// TwinCAT 3 PLC project TE1108
// ProgramVersion: 3.1.4026.22
// libraries:
//   Tc2_EtherCAT, * (Beckhoff Automation GmbH)
//   Tc2_IoFunctions, * (Beckhoff Automation GmbH)
//   Tc2_Standard, * (Beckhoff Automation GmbH)
//   Tc2_System, * (Beckhoff Automation GmbH)
//   Tc2_Utilities, * (Beckhoff Automation GmbH)
//   Tc3_Module, * (Beckhoff Automation GmbH)
// project tree:
//   DUTs/COMPONENTS/GENERIC/ ST_GeneralStationCMD.TcDUT (not stored), ST_StationStatus.TcDUT (not stored)
//   DUTs/COMPONENTS/HEIGHT TEST/ ST_HeightTest.TcDUT (not stored), ST_HeightTest_CMD.TcDUT (not stored), ST_ProbesSettings.TcDUT, E_HeightTest_State.TcDUT (not stored), ST_HeightTest_CycleData.TcDUT (not stored)
//   DUTs/COMPONENTS/LEAK TESTER/ ST_LeakTester.TcDUT (not stored), ST_LeakTester_CMD.TcDUT (not stored), E_LeakTester_State.TcDUT (not stored), ST_LeakTester_CycleData.TcDUT (not stored)
//   DUTs/COMPONENTS/MAIN CYLINDER/ ST_ProcessCylinder.TcDUT (not stored), E_ProcessCylinder_State.TcDUT (not stored), ST_ProcessCylinder_CMD.TcDUT (not stored)
//   DUTs/COMPONENTS/PROCESS DOOR/ E_ProcessDoor_State.TcDUT (not stored), ST_ProcessDoor.TcDUT (not stored), ST_ProcessDoor_CMD.TcDUT (not stored)
//   DUTs/COMPONENTS/SLIDE NEST/ E_SlideNest_State.TcDUT (not stored), ST_SlideNest.TcDUT (not stored), ST_SlideNest_CMD.TcDUT (not stored)
//   DUTs/HMI/ ST_Animations.TcDUT (not stored), ST_StatisticsHMI.TcDUT (not stored), ST_StatusBanner.TcDUT (not stored), ST_Timers.TcDUT (not stored)
//   DUTs/IO/CARDS/ ST_EL1918_C.TcDUT (not stored), ST_EL3058.TcDUT (not stored), ST_EL1918_A.TcDUT (not stored), ST_EL1918_B.TcDUT (not stored), ST_EL2904.TcDUT (not stored), ST_EL6910.TcDUT (not stored), ST_EL6633.TcDUT (not stored), ST_EL9410.TcDUT (not stored), ST_K1100.TcDUT (not stored), ST_EL6070.TcDUT (not stored), ST_Terminal_Info.TcDUT (not stored), ST_EL1809.TcDUT, ST_EL2809_A.TcDUT
//   DUTs/IO/LEAK_TESTERS/ ST_General_LeakTester_I_O.TcDUT (not stored), st_i28General_I_O.TcDUT (not stored), st_i28LasResult.TcDUT (not stored), st_i28LiveMeasurement.TcDUT (not stored)
//   DUTs/IO/PROBES/ ST_ProbesSet.TcDUT (not stored), ST_Probes_I_O.TcDUT (not stored)
//   DUTs/MASTER/ E_MachineState.TcDUT (not stored), ST_ButtonsLamps.TcDUT (not stored), ST_MachineStatus.TcDUT (not stored), ST_MasterCTRL.TcDUT (not stored), ST_Puls.TcDUT (not stored)
//   DUTs/MASTER/log_CSV/ ST_TableCycleData.TcDUT (not stored), ST_UserLog.TcDUT (not stored), ST_CycleData.TcDUT (not stored)
//   DUTs/MASTER/PROCESS CYCLES/ E_General_ProcessCycle.TcDUT
//   DUTs/PDFMaker/ ST_EventsPDF.TcDUT (not stored), ST_EventsPdfConstants.TcDUT (not stored), ST_JavasCriptPDF.TcDUT (not stored), ST_PDFMaker.TcDUT (not stored)
//   DUTs/ ST_SafeOutputsReading.TcDUT (not stored), ST_TwinSAFE.TcDUT (not stored)
//   DUTs/USER_ALARMS_EVENTS/EVENTS/ ST_ActiveEvents.TcDUT (not stored), ST_EventsAssigment.TcDUT (not stored), ST_EventsAssigmentGeneral.TcDUT (not stored), ST_EventsHistory.TcDUT (not stored), ST_EVENT.TcDUT (not stored), ST_StationEvents.TcDUT (not stored)
//   DUTs/USER_ALARMS_EVENTS/ ST_UserLogHMI.TcDUT (not stored)
//   GVLs/ GVL_Constants.TcGVL (not stored), GVL_HMI.TcGVL, GVL_IO.TcGVL (not stored), GVL_Master.TcGVL, GVL_Persistent.TcGVL (not stored), GVL_Stations.TcGVL
//   / PlcTask.TcTTO (not stored)
//   POUs/A_MASTER/ A_1_PRG_Main_Master.TcPOU, A_2_PRG_MachineCtrl.TcPOU, A_3_PRG_FaultHandling.TcPOU
//   POUs/B_STATIONS/B_1_LEAK_TEST/ B_1_1_PRG_Master_Leak_Test.TcPOU
//   POUs/B_STATIONS/B_2_HEIGHT_TEST/ B_2_1_PRG_Master_Height_Test.TcPOU (not stored)
//   POUs/B_STATIONS/B_4_PROCESS_CYLINDER__SLIDE_DOOR_SLIDE_NEST/ B_4_1_PRG_Master_ProcessCylinder.TcPOU, B_4_2_PRG_Master_ProcessDoor.TcPOU, B_4_3_PRG_Master_SlideNest.TcPOU
//   POUs/C_HMI/ C_1_PRG_MainHMI.TcPOU
//   POUs/D_CSV/ D_1_PRG_CycleDataCSV.TcPOU (not stored)
//   POUs/ MAIN.TcPOU (not stored)
//   POUs/Utilities/ FB_EventsManager.TcPOU (not stored), FB_PDFMaker.TcPOU (not stored), FB_Scale.TcPOU (not stored), FB_UserLog.TcPOU (not stored), FB_Pulse.TcPOU (not stored), FB_TerminalInfo.TcPOU (not stored), FB_TimeControl.TcPOU (not stored), PRG_Puls.TcPOU (not stored)
// real-time tasks:
//   TASK PlcTask: cycle T#10ms, priority 20, ADS port 350
// I/O:
//   DEVICE Device1(EtherCAT), AmsNetId 192.168.7.156.4.1
//     Term 1 (EK1100) [EK1100 EtherCAT Coupler (2A E-Bus)]
//       Term 2 (EL6070-0033) [EL6070-0033 1Ch. Licence key terminal, individual licences]
//       Term 3 (EL6910) [EL6910, TwinSAFE PLC]
//       Term 4 (EL1918) [EL1918, 8Ch. Safety Input 24V, TwinSAFE]
//         modules: Module 1 (FSOE), Module 2 (FSLOGIC)
//       Term 5 (EL1918) [EL1918, 8Ch. Safety Input 24V, TwinSAFE]
//         modules: Module 1 (FSOE), Module 2 (FSLOGIC)
//       Term 6 (EL2904) [EL2904, 4 Ch. Safety Output 24V, 0.5A, TwinSAFE]
//         modules: Module 1 (FSOES), Module 2 (DO)
//       Term 7 (EL9410) [EL9410 E-Bus Power Supplier  (Diagnostics)]
//       Term 8 (EL1809) [EL1809 16Ch. Dig. Input 24V, 3ms]
//       Term 9 (EL2809) [EL2809 16Ch. Dig. Output 24V, 0.5A]
//       Term 10 (EL3058) [EL3058 8Ch. Ana. Input 4-20mA]
//       Term 11(EL1918) [EL1918, 8Ch. Safety Input 24V, TwinSAFE]
//         modules: Module 1 (FSOE), Module 2 (FSLOGIC)
//       Term 12 (EL6633) [EL6633 PROFINET IO Controller]
//       Term 13 (EL9011) [EL9011 End Terminal]
//     Box 21 (DL-EC1A) [DL-EC1A]
//   DEVICE Profinet1 (EL6633), AmsNetId 192.168.7.156.2.1
//     fpc1 [Cincinnati Test Systems 1-port Device 00210]
//       modules: Term 1 (DAP Module), Term 2 (PLC Input), Term 3 (PLC Output  )
//     fpc2 [Cincinnati Test Systems 1-port Device 00210]
//       modules: Term 4 (DAP Module), Term 5 (PLC Input), Term 6 (PLC Output  )
// variable links:
//   Device1(EtherCAT) <-> Device1(EtherCAT)/Term 1 (EK1100)/Term 11(EL1918)
//     Term 1 (EK1100)/Term 3 (EL6910)/ConnectionInputs/Message_38 TxPDO <-> Module 1 (FSOE)/FSoE Outputs/FSOE
//     Term 1 (EK1100)/Term 3 (EL6910)/ConnectionOutputs/Message_38 RxPDO <-> Module 1 (FSOE)/FSoE Inputs/FSOE
//   Device1(EtherCAT) <-> Device1(EtherCAT)/Term 1 (EK1100)/Term 4 (EL1918)
//     Term 1 (EK1100)/Term 3 (EL6910)/ConnectionInputs/Message_8 TxPDO <-> Module 1 (FSOE)/FSoE Outputs/FSOE
//     Term 1 (EK1100)/Term 3 (EL6910)/ConnectionOutputs/Message_8 RxPDO <-> Module 1 (FSOE)/FSoE Inputs/FSOE
//   Device1(EtherCAT) <-> Device1(EtherCAT)/Term 1 (EK1100)/Term 5 (EL1918)
//     Term 1 (EK1100)/Term 3 (EL6910)/ConnectionInputs/Message_9 TxPDO <-> Module 1 (FSOE)/FSoE Outputs/FSOE
//     Term 1 (EK1100)/Term 3 (EL6910)/ConnectionOutputs/Message_9 RxPDO <-> Module 1 (FSOE)/FSoE Inputs/FSOE
//   Device1(EtherCAT) <-> Device1(EtherCAT)/Term 1 (EK1100)/Term 6 (EL2904)
//     Term 1 (EK1100)/Term 3 (EL6910)/ConnectionInputs/Message_10 TxPDO <-> Module 1 (FSOES)/RxPDO/FSOE
//     Term 1 (EK1100)/Term 3 (EL6910)/ConnectionOutputs/Message_10 RxPDO <-> Module 1 (FSOES)/TxPDO/FSOE
//   TE1108/TE1108 Instance <-> Device1(EtherCAT)/Box 21 (DL-EC1A)
//     PlcTask Inputs/GVL_IO.Probes.bGeneralError <-> Status of System/Error Status
//     PlcTask Inputs/GVL_IO.Probes.stProbesSet[1].abProbeError[1] <-> ID01 Status/ID01 Error Status
//     PlcTask Inputs/GVL_IO.Probes.stProbesSet[1].abProbeError[2] <-> ID02 Status/ID02 Error Status
//     PlcTask Inputs/GVL_IO.Probes.stProbesSet[1].abProbeError[3] <-> ID03 Status/ID03 Error Status
//     PlcTask Inputs/GVL_IO.Probes.stProbesSet[1].abProbeError[4] <-> ID04 Status/ID04 Error Status
//     PlcTask Inputs/GVL_IO.Probes.stProbesSet[2].abProbeError[1] <-> ID05 Status/ID05 Error Status
//     PlcTask Inputs/GVL_IO.Probes.stProbesSet[2].abProbeError[2] <-> ID06 Status/ID06 Error Status
//     PlcTask Inputs/GVL_IO.Probes.stProbesSet[2].abProbeError[3] <-> ID07 Status/ID07 Error Status
//     PlcTask Inputs/GVL_IO.Probes.stProbesSet[2].abProbeError[4] <-> ID08 Status/ID08 Error Status
//     PlcTask Inputs/GVL_IO.Probes.stProbesSet[1].anRawMeasurement[1] <-> ID01 Current Value/ID01 Current Value (P.V.)
//     PlcTask Inputs/GVL_IO.Probes.stProbesSet[1].anRawMeasurement[2] <-> ID02 Current Value/ID02 Current Value (P.V.)
//     PlcTask Inputs/GVL_IO.Probes.stProbesSet[1].anRawMeasurement[3] <-> ID03 Current Value/ID03 Current Value (P.V.)
//     PlcTask Inputs/GVL_IO.Probes.stProbesSet[1].anRawMeasurement[4] <-> ID04 Current Value/ID04 Current Value (P.V.)
//     PlcTask Inputs/GVL_IO.Probes.stProbesSet[2].anRawMeasurement[1] <-> ID05 Current Value/ID05 Current Value (P.V.)
//     PlcTask Inputs/GVL_IO.Probes.stProbesSet[2].anRawMeasurement[2] <-> ID06 Current Value/ID06 Current Value (P.V.)
//     PlcTask Inputs/GVL_IO.Probes.stProbesSet[2].anRawMeasurement[3] <-> ID07 Current Value/ID07 Current Value (P.V.)
//     PlcTask Inputs/GVL_IO.Probes.stProbesSet[2].anRawMeasurement[4] <-> ID08 Current Value/ID08 Current Value (P.V.)
//     PlcTask Inputs/GVL_IO.Probes.stTerminalInfo.nTerminal_State <-> InfoData/State
//     PlcTask Outputs/GVL_IO.Probes.abPresetProbe <-> Input Request 1/Request 1
//   TE1108/TE1108 Instance <-> Device1(EtherCAT)/Term 1 (EK1100)
//     PlcTask Inputs/GVL_IO.dw_T01_EK1100.stTerminalInfo.nTerminal_State <-> InfoData/State
//   TE1108/TE1108 Instance <-> Device1(EtherCAT)/Term 1 (EK1100)/Term 10 (EL3058)
//     PlcTask Inputs/GVL_IO.dw_T10_EL3058.iMainPressure <-> AI Standard Channel 1/Value
//     PlcTask Inputs/GVL_IO.dw_T10_EL3058.stTerminalInfo.nTerminal_State <-> InfoData/State
//   TE1108/TE1108 Instance <-> Device1(EtherCAT)/Term 1 (EK1100)/Term 11(EL1918)
//     PlcTask Inputs/GVL_IO.dw_T11_EL1918.iD3ProcessCylinderFeedback <-> Module 1 (FSOE)/FSoE Inputs/FSOE/FSIN Module 3.Input
//     PlcTask Inputs/GVL_IO.dw_T11_EL1918.iD3ProcessCylinderRetracted1 <-> Module 1 (FSOE)/FSoE Inputs/FSOE/FSIN Module 1.Input
//     PlcTask Inputs/GVL_IO.dw_T11_EL1918.iD3ProcessCylinderRetracted2 <-> Module 1 (FSOE)/FSoE Inputs/FSOE/FSIN Module 2.Input
//     PlcTask Inputs/GVL_IO.dw_T11_EL1918.stTerminalInfo.nTerminal_State <-> InfoData/State
//   TE1108/TE1108 Instance <-> Device1(EtherCAT)/Term 1 (EK1100)/Term 12 (EL6633)
//     PlcTask Inputs/GVL_IO.dw_T12_EL6633.stTerminalInfo.nTerminal_State <-> InfoData/State
//   TE1108/TE1108 Instance <-> Device1(EtherCAT)/Term 1 (EK1100)/Term 2 (EL6070-0033)
//     PlcTask Inputs/GVL_IO.dw_T02_EL6070.stTerminalInfo.nTerminal_State <-> InfoData/State
//   TE1108/TE1108 Instance <-> Device1(EtherCAT)/Term 1 (EK1100)/Term 3 (EL6910)
//     PlcTask Inputs/GVL_IO.dw_T03_EL6910.stTerminalInfo.nTerminal_State <-> InfoData/State
//     PlcTask Inputs/GVL_IO.stTwinSAFE.qAirErrorSignal <-> StandardInputs/TwinSafeGroup1.AirErrorSignal_59
//     PlcTask Inputs/GVL_IO.stTwinSAFE.qAirPressureAbove <-> StandardInputs/TwinSafeGroup1.AirPressureAbove_26
//     PlcTask Inputs/GVL_IO.stTwinSAFE.qAirPressureBelow <-> StandardInputs/TwinSafeGroup1.AirPressureBelow_25
//     PlcTask Inputs/GVL_IO.stTwinSAFE.qAirPressureOK <-> StandardInputs/TwinSafeGroup1.AirPressureOK_41
//     PlcTask Inputs/GVL_IO.stTwinSAFE.qComError <-> StandardInputs/TwinSafeGroup1.COMError_74
//     PlcTask Inputs/GVL_IO.stTwinSAFE.qE_StopPressed <-> StandardInputs/TwinSafeGroup1.E_StopPressed_32
//     PlcTask Inputs/GVL_IO.stTwinSAFE.qFBError <-> StandardInputs/TwinSafeGroup1.FBError_73
//     PlcTask Inputs/GVL_IO.stTwinSAFE.qMainDoorOpenned <-> StandardInputs/TwinSafeGroup1.DoorOpenned_68
//     PlcTask Inputs/GVL_IO.stTwinSAFE.qMainDoorUnsafe <-> StandardInputs/TwinSafeGroup1.MainDoorUnsafe_49
//     PlcTask Inputs/GVL_IO.stTwinSAFE.qOtherError <-> StandardInputs/TwinSafeGroup1.OtherError_75
//     PlcTask Inputs/GVL_IO.stTwinSAFE.qProcessCylinderRetracted <-> StandardInputs/TwinSafeGroup1.ProcessCylinderRetracted_60
//     PlcTask Inputs/GVL_IO.stTwinSAFE.qProcessCylinderUnsafe <-> StandardInputs/TwinSafeGroup1.ProcessCylinderUnsafe_54
//     PlcTask Inputs/GVL_IO.stTwinSAFE.qProcessDoorUnSafe <-> StandardInputs/TwinSafeGroup1.ProcessDoorUnsafe_34
//     PlcTask Inputs/GVL_IO.stTwinSAFE.qSafetyOk <-> StandardInputs/TwinSafeGroup1.SafetyOK_30
//     PlcTask Inputs/GVL_IO.stTwinSAFE.qSystemSafe <-> StandardInputs/TwinSafeGroup1.SystemSafe_72
//     PlcTask Inputs/GVL_IO.stTwinSAFE.qTwoHandsSafe <-> StandardInputs/TwinSafeGroup1.TwoHandsSafe_77
//     PlcTask Inputs/GVL_IO.stTwinSAFE.qTwoHandsUnsafe <-> StandardInputs/TwinSafeGroup1.TwoHandsUnsafe_35
//     PlcTask Outputs/GVL_IO.stTwinSAFE.iAirPressureMaxValue <-> StandardOutputs/TwinSafeGroup1.AirPressureMaxVal_23
//     PlcTask Outputs/GVL_IO.stTwinSAFE.iAirPressureMinValue <-> StandardOutputs/TwinSafeGroup1.AirPressureMinVal_22
//     PlcTask Outputs/GVL_IO.stTwinSAFE.iAirSupplyMeasurement <-> StandardOutputs/TwinSafeGroup1.AirSupplyMeasurement_19
//     PlcTask Outputs/GVL_IO.stTwinSAFE.iMachineHoming_Manual <-> StandardOutputs/TwinSafeGroup1.MachineHoming_Manual_78
//     PlcTask Outputs/GVL_IO.stTwinSAFE.iMachineStopped <-> StandardOutputs/TwinSafeGroup1.MachineStopped_70
//     PlcTask Outputs/GVL_IO.stTwinSAFE.iProcessDoorClosedCondition <-> StandardOutputs/TwinSafeGroup1.ProcessDoorClosedCondition_16
//     PlcTask Outputs/GVL_IO.stTwinSAFE.iProcessDoorClosing <-> StandardOutputs/TwinSafeGroup1.ProcessDoor Closing_29
//     PlcTask Outputs/GVL_IO.stTwinSAFE.iRunSafety <-> StandardOutputs/TwinSafeGroup1.RunSafety_69
//     PlcTask Outputs/GVL_IO.stTwinSAFE.iSafetyErrorAcknowledge <-> StandardOutputs/TwinSafeGroup1.SafetyErrorAcknowledge_55
//   TE1108/TE1108 Instance <-> Device1(EtherCAT)/Term 1 (EK1100)/Term 4 (EL1918)
//     PlcTask Inputs/GVL_IO.dw_T04_EL1918.iD1MainDoorFB <-> Module 1 (FSOE)/FSoE Inputs/FSOE/FSIN Module 6.Input
//     PlcTask Inputs/GVL_IO.dw_T04_EL1918.iD1MainDoorLocked1 <-> Module 1 (FSOE)/FSoE Inputs/FSOE/FSIN Module 4.Input
//     PlcTask Inputs/GVL_IO.dw_T04_EL1918.iD1MainDoorLocked2 <-> Module 1 (FSOE)/FSoE Inputs/FSOE/FSIN Module 5.Input
//     PlcTask Inputs/GVL_IO.dw_T04_EL1918.iEStopChannel1 <-> Module 1 (FSOE)/FSoE Inputs/FSOE/FSIN Module 1.Input
//     PlcTask Inputs/GVL_IO.dw_T04_EL1918.iEStopChannel2 <-> Module 1 (FSOE)/FSoE Inputs/FSOE/FSIN Module 2.Input
//     PlcTask Inputs/GVL_IO.dw_T04_EL1918.iFestoMS6DumpValveFB <-> Module 1 (FSOE)/FSoE Inputs/FSOE/FSIN Module 8.Input
//     PlcTask Inputs/GVL_IO.dw_T04_EL1918.iFestoMS6ValveFB <-> Module 1 (FSOE)/FSoE Inputs/FSOE/FSIN Module 7.Input
//     PlcTask Inputs/GVL_IO.dw_T04_EL1918.iResetButton <-> Module 1 (FSOE)/FSoE Inputs/FSOE/FSIN Module 3.Input
//     PlcTask Inputs/GVL_IO.dw_T04_EL1918.stTerminalInfo.nTerminal_State <-> InfoData/State
//   TE1108/TE1108 Instance <-> Device1(EtherCAT)/Term 1 (EK1100)/Term 5 (EL1918)
//     PlcTask Inputs/GVL_IO.dw_T05_EL1918.iLeftTouchButtonNC <-> Module 1 (FSOE)/FSoE Inputs/FSOE/FSIN Module 1.Input
//     PlcTask Inputs/GVL_IO.dw_T05_EL1918.iLeftTouchButtonNO <-> Module 1 (FSOE)/FSoE Inputs/FSOE/FSIN Module 3.Input
//     PlcTask Inputs/GVL_IO.dw_T05_EL1918.iProcessDoorClosed1 <-> Module 1 (FSOE)/FSoE Inputs/FSOE/FSIN Module 5.Input
//     PlcTask Inputs/GVL_IO.dw_T05_EL1918.iProcessDoorClosed2 <-> Module 1 (FSOE)/FSoE Inputs/FSOE/FSIN Module 6.Input
//     PlcTask Inputs/GVL_IO.dw_T05_EL1918.iProcessDoorFB <-> Module 1 (FSOE)/FSoE Inputs/FSOE/FSIN Module 7.Input
//     PlcTask Inputs/GVL_IO.dw_T05_EL1918.iRightTouchButtonNC <-> Module 1 (FSOE)/FSoE Inputs/FSOE/FSIN Module 2.Input
//     PlcTask Inputs/GVL_IO.dw_T05_EL1918.iRightTouchButtonNO <-> Module 1 (FSOE)/FSoE Inputs/FSOE/FSIN Module 4.Input
//     PlcTask Inputs/GVL_IO.dw_T05_EL1918.stTerminalInfo.nTerminal_State <-> InfoData/State
//   TE1108/TE1108 Instance <-> Device1(EtherCAT)/Term 1 (EK1100)/Term 6 (EL2904)
//     PlcTask Inputs/GVL_IO.dw_T06_EL2904.stTerminalInfo.nTerminal_State <-> InfoData/State
//   TE1108/TE1108 Instance <-> Device1(EtherCAT)/Term 1 (EK1100)/Term 7 (EL9410)
//     PlcTask Inputs/GVL_IO.dw_T07_EL9410.stTerminalInfo.nTerminal_State <-> InfoData/State
//   TE1108/TE1108 Instance <-> Device1(EtherCAT)/Term 1 (EK1100)/Term 8 (EL1809)
//     PlcTask Inputs/GVL_IO.dw_T08_EL1809.iPartPresentNest1 <-> Channel 5/Input
//     PlcTask Inputs/GVL_IO.dw_T08_EL1809.iPartPresentNest2 <-> Channel 6/Input
//     PlcTask Inputs/GVL_IO.dw_T08_EL1809.iProcessCylinderExtended <-> Channel 10/Input
//     PlcTask Inputs/GVL_IO.dw_T08_EL1809.iPuckSensorDown <-> Channel 16/Input
//     PlcTask Inputs/GVL_IO.dw_T08_EL1809.iPuckSensorUp <-> Channel 15/Input
//     PlcTask Inputs/GVL_IO.dw_T08_EL1809.iRejectSensor <-> Channel 11/Input
//     PlcTask Inputs/GVL_IO.dw_T08_EL1809.iSlideNestExtended <-> Channel 7/Input
//     PlcTask Inputs/GVL_IO.dw_T08_EL1809.iSlideNestRetracted <-> Channel 8/Input
//     PlcTask Inputs/GVL_IO.dw_T08_EL1809.iStartButoon <-> Channel 1/Input
//     PlcTask Inputs/GVL_IO.dw_T08_EL1809.iStopButton <-> Channel 2/Input
//     PlcTask Inputs/GVL_IO.dw_T08_EL1809.iUP_OK <-> Channel 3/Input
//     PlcTask Inputs/GVL_IO.dw_T08_EL1809.iUS_OK <-> Channel 4/Input
//     PlcTask Inputs/GVL_IO.dw_T08_EL1809.stTerminalInfo.nTerminal_State <-> InfoData/State
//   TE1108/TE1108 Instance <-> Device1(EtherCAT)/Term 1 (EK1100)/Term 9 (EL2809)
//     PlcTask Inputs/GVL_IO.dw_T09_EL2809.stTerminalInfo.nTerminal_State <-> InfoData/State
//     PlcTask Outputs/GVL_IO.dw_T09_EL2809.qBottomSealer <-> Channel 14/Output
//     PlcTask Outputs/GVL_IO.dw_T09_EL2809.qCloseProcessDoor <-> Channel 4/Output
//     PlcTask Outputs/GVL_IO.dw_T09_EL2809.qExtendProcessCylinder <-> Channel 6/Output
//     PlcTask Outputs/GVL_IO.dw_T09_EL2809.qExtendSlideNest <-> Channel 13/Output
//     PlcTask Outputs/GVL_IO.dw_T09_EL2809.qIndicatorLED1_Green <-> Channel 9/Output
//     PlcTask Outputs/GVL_IO.dw_T09_EL2809.qIndicatorLED2_Green <-> Channel 11/Output
//     PlcTask Outputs/GVL_IO.dw_T09_EL2809.qIndicatorLED1_Red <-> Channel 8/Output
//     PlcTask Outputs/GVL_IO.dw_T09_EL2809.qIndicatorLED2_Red <-> Channel 10/Output
//     PlcTask Outputs/GVL_IO.dw_T09_EL2809.qOpenProcessDoor <-> Channel 3/Output
//     PlcTask Outputs/GVL_IO.dw_T09_EL2809.qPanelLightLED <-> Channel 7/Output
//     PlcTask Outputs/GVL_IO.dw_T09_EL2809.qPuckLockerPinCommand <-> Channel 16/Output
//     PlcTask Outputs/GVL_IO.dw_T09_EL2809.qResetButtonLED <-> Channel 2/Output
//     PlcTask Outputs/GVL_IO.dw_T09_EL2809.qRetractProcessCylinder <-> Channel 5/Output
//     PlcTask Outputs/GVL_IO.dw_T09_EL2809.qRetractSlideNest <-> Channel 12/Output
//     PlcTask Outputs/GVL_IO.dw_T09_EL2809.qStartButtonLED <-> Channel 1/Output
//     PlcTask Outputs/GVL_IO.dw_T09_EL2809.qTopSealer <-> Channel 15/Output
//   TE1108/TE1108 Instance <-> Profinet1 (EL6633)/fpc1
//     PlcTask Inputs/GVL_IO.LeakTester1_IO.sti28General_I_O.bInstrumentReady <-> API/Term 2 (PLC Input)/Subterm 4 (Instrument Status)/Inputs/Instrument Status/Instrument_Ready
//     PlcTask Inputs/GVL_IO.LeakTester1_IO.sti28General_I_O.bMalfunction <-> API/Term 2 (PLC Input)/Subterm 4 (Instrument Status)/Inputs/Instrument Status/Malfunction
//     PlcTask Inputs/GVL_IO.LeakTester1_IO.sti28General_I_O.bProgramAccept <-> API/Term 2 (PLC Input)/Subterm 4 (Instrument Status)/Inputs/Instrument Status/Program_Accept
//     PlcTask Inputs/GVL_IO.LeakTester1_IO.sti28General_I_O.bProgramReject <-> API/Term 2 (PLC Input)/Subterm 4 (Instrument Status)/Inputs/Instrument Status/Program_Reject
//     PlcTask Inputs/GVL_IO.LeakTester1_IO.sti28General_I_O.bTestActiveLiveData <-> API/Term 2 (PLC Input)/Subterm 4 (Instrument Status)/Inputs/Instrument Status/Test_Active_Live_Data
//     PlcTask Outputs/GVL_IO.LeakTester1_IO.sti28General_I_O.bReset <-> API/Term 3 (PLC Output  )/Subterm 7 (Instrument Control )/Outputs/Instrument Control/Reset
//     PlcTask Outputs/GVL_IO.LeakTester1_IO.sti28General_I_O.bStart <-> API/Term 3 (PLC Output  )/Subterm 7 (Instrument Control )/Outputs/Instrument Control/Start
//     PlcTask Outputs/GVL_IO.LeakTester1_IO.sti28General_I_O.bStop <-> API/Term 3 (PLC Output  )/Subterm 7 (Instrument Control )/Outputs/Instrument Control/Stop
//   TE1108/TE1108 Instance <-> Profinet1 (EL6633)/fpc2
//     PlcTask Inputs/GVL_IO.LeakTester2_IO.sti28General_I_O.bInstrumentReady <-> API/Term 5 (PLC Input)/Subterm 12 (Instrument Status)/Inputs/Instrument Status/Instrument_Ready
//     PlcTask Inputs/GVL_IO.LeakTester2_IO.sti28General_I_O.bMalfunction <-> API/Term 5 (PLC Input)/Subterm 12 (Instrument Status)/Inputs/Instrument Status/Malfunction
//     PlcTask Inputs/GVL_IO.LeakTester2_IO.sti28General_I_O.bProgramAccept <-> API/Term 5 (PLC Input)/Subterm 12 (Instrument Status)/Inputs/Instrument Status/Program_Accept
//     PlcTask Inputs/GVL_IO.LeakTester2_IO.sti28General_I_O.bProgramReject <-> API/Term 5 (PLC Input)/Subterm 12 (Instrument Status)/Inputs/Instrument Status/Program_Reject
//     PlcTask Inputs/GVL_IO.LeakTester2_IO.sti28General_I_O.bTestActiveLiveData <-> API/Term 5 (PLC Input)/Subterm 12 (Instrument Status)/Inputs/Instrument Status/Test_Active_Live_Data
//     PlcTask Outputs/GVL_IO.LeakTester2_IO.sti28General_I_O.bReset <-> API/Term 6 (PLC Output  )/Subterm 15 (Instrument Control )/Outputs/Instrument Control/Reset
//     PlcTask Outputs/GVL_IO.LeakTester2_IO.sti28General_I_O.bStart <-> API/Term 6 (PLC Output  )/Subterm 15 (Instrument Control )/Outputs/Instrument Control/Start
//     PlcTask Outputs/GVL_IO.LeakTester2_IO.sti28General_I_O.bStop <-> API/Term 6 (PLC Output  )/Subterm 15 (Instrument Control )/Outputs/Instrument Control/Stop

// ---- DUTs/COMPONENTS/HEIGHT TEST/ST_ProbesSettings.TcDUT
TYPE ST_ProbesSettings :
STRUCT
	
	anDistanceCalibrationBlock			: ARRAY [1..3] OF REAL;	
	nDistanceOffset1					: ARRAY [1..3] OF REAL; 
	nDistanceOffset2					: ARRAY [1..3] OF REAL;	
	anExpectedDistances					: ARRAY [1..3] OF REAL;
	anHeightSetByCalibration1			: ARRAY [1..4] OF REAL;	
	anHeightSetByCalibration2			: ARRAY [1..4] OF REAL;	
	anTolerances						: ARRAY [1..3] OF REAL;	


END_STRUCT
END_TYPE

// ---- DUTs/IO/CARDS/ST_EL1809.TcDUT
TYPE ST_EL1809 :
STRUCT
	//--------------------------------------------------------------------------------------------------------
	sTerminalName                                           :   STRING(200):= 'EL1809 | 16-Channel Digital Input';
    //============================================================================================================================	
	// TERMINAL - EL1809 16-Channel Digital Input Terminal (Term 8)	
	iStartButoon                			AT %I*			: 	BOOL;	// EL1809 channel 1
	iStopButton                   			AT %I*			: 	BOOL;	// EL1809 channel 2
	iUP_OK        							AT %I*	 		: 	BOOL;	// EL1809 channel 3
	iUS_OK		   							AT %I*	 		: 	BOOL;	// EL1809 channel 4
	iPartPresentNest1         				AT %I*	 		: 	BOOL;	// EL1809 channel 5 		     			
	iPartPresentNest2 						AT %I*			: 	BOOL;	// EL1809 channel 6
	iSlideNestRetracted    					AT %I*          :   BOOL;   // EL1809 channel 7 
    iSlideNestExtended         				AT %I*          :   BOOL;   // EL1809 channel 8
    iEL1809_Ch9           					AT %I*          :   BOOL;   // EL1809 channel 9
	iProcessCylinderExtended              	AT %I*          :   BOOL;   // EL1809 channel 10
	iRejectSensor              				AT %I*          :   BOOL;   // EL1809 channel 11
	iEL1809_Ch12			              	AT %I*          :   BOOL;   // EL1809 channel 12	   
	iEL1809_Ch13         		   			AT %I*	 		: 	BOOL;	// EL1809 channel 13   
	iEL1809_Ch14       						AT %I*	 		: 	BOOL;	// EL1809 channel 14 
	iEL1809_Ch15							AT %I*			: 	BOOL;	// EL1809 channel 15  
	iEL1809_Ch16							AT %I*	 		: 	BOOL;	// EL1809 channel 16  	
	
	stTerminalInfo											: 	ST_Terminal_Info;

END_STRUCT
END_TYPE

// ---- DUTs/IO/CARDS/ST_EL2809_A.TcDUT
TYPE ST_EL2809_A :
STRUCT
	//--------------------------------------------------------------------------------------------------------
	sTerminalName                                           :   STRING(200):= 'EL2809 | 16-Channel Digital Output';
	//=============================================================================================================
	// TERMINAL - EL2809	16-Channel Digital Output Terminal	 (Term 9)
	qStartButtonLED							AT %Q*			: 	BOOL;	// EL2809 channel 1
	qResetButtonLED							AT %Q* 			: 	BOOL;	// EL2809 channel 2
	qOpenProcessDoor             			AT %Q*	 		: 	BOOL;	// EL2809 channel 3 			
	qCloseProcessDoor      					AT %Q*	 		: 	BOOL;	// EL2809 channel 4 
	qRetractProcessCylinder  				AT %Q*	 		: 	BOOL;	// EL2809 channel 5
	qExtendProcessCylinder	 				AT %Q*	 		: 	BOOL;	// EL2809 channel 6 	
	qPanelLightLED         		    		AT %Q*			: 	BOOL;	// EL2809 channel 7	
	qIndicatorLED1_Red						AT %Q*	 		: 	BOOL;	// EL2809 channel 8	
	qIndicatorLED1_Green                 	AT %Q*          :   BOOL;   // EL2809 channel 9
	qIndicatorLED2_Red             			AT %Q*          :   BOOL;   // EL2809 channel 10   	
	qIndicatorLED2_Green     				AT %Q*	 		: 	BOOL;	// EL2809 channel 11	
	qRetractSlideNest   					AT %Q*	 		: 	BOOL;	// EL2809 channel 12 
    qExtendSlideNest			        	AT %Q*	 		: 	BOOL;	// EL2809 channel 13 
	qBottomSealer            				AT %Q*	 		: 	BOOL;	// EL2809 channel 14 
	qTopSealer								AT %Q*	 		: 	BOOL;	// EL2809 channel 15 
    qPuckLockerPinCommand  	        		AT %Q*	 		: 	BOOL;	// EL2809 channel 16
	
	stTerminalInfo											: 	ST_Terminal_Info;
	
END_STRUCT
END_TYPE

// ---- DUTs/MASTER/PROCESS CYCLES/E_General_ProcessCycle.TcDUT
{attribute 'qualified_only'}
{attribute 'strict'}
TYPE E_General_ProcessCycle :
(
	
IDLE							,
CLOSE_PROCESS_DOOR				,
WAIT_CLOSE_PROCESS_DOOR			,
OPEN_PROCESS_DOOR				,
WAIT_OPEN_PROCESS_DOOR			,
PRE_RETRACT_PROCESS_CYLINDER		,	//Renan added - Buglist n13 - 08Jul26
WAIT_PRE_RETRACT_PROCESS_CYLINDER	, 	//Renan added - Buglist n13 - 08Jul26
EXTEND_PROCESS_CYLINDER			,
WAIT_EXTEND_PROCESS_CYLINDER	,
RETRACT_PROCESS_CYLINDER		,
WAIT_RETRACT_PROCESS_CYLINDER	,
RETRACT_MIDDLE_PROCESS_CYLINDER		,
WAIT_RETRACT_MIDDLE_PROCESS_CYLINDER	,
MOVE_NEST_TO_RIGHT				,
WAIT_MOVE_NEST_TO_RIGHT			,
MOVE_NEST_TO_LEFT				,
WAIT_MOVE_NEST_TO_LEFT			,
LEAK_TEST						,
WAIT_LEAK_TEST					,
HEIGHT_TEST						,
WAIT_HEIGHT_TEST				,
WAIT_TO_SAVE_DATA				,
WAIT_RESULTS					,
RESULTS							,
SAVE_DATA						,
SAVE_DATA2						,
CSV_NEST1						,
CSV_NEST2						,
WAIT_REJECT_PART				,
REJECT_CHUTE_FULL				,
PUCK_DEFINITION						,
NEST_CLEARING						,

RESET_ALL_CMD						

);
END_TYPE

// ---- GVLs/GVL_HMI.TcGVL
VAR_GLOBAL
////////////////////////////////////////:	///////////////////////////////////////////////////
/////////////////////////////////////////////////////////////////////////////////////GENERIC/////////////////////////////////////////////////////////////////////////////////////

	bQuitHMI							: BOOL;
	bShutDown							: BOOL;
	stStatusBanner						: ST_StatusBanner;
	nPopUp								: DINT;
	
	bPartPresent						: ARRAY [0..1] OF BOOL;
	
	bRejectPartDialog					: ARRAY [0..2] OF BOOL;
	bOpenRejectDialog					: BOOL;
	bLightsOnOff						: BOOL;
	
	bHMIAlive							: BOOL;
	tonHMIAliveOn						: TON;
	tonHMIAliveOff						: TON;
	bOutHMI								: BOOL;
	
/////////////////////////////////////////////////////////////////////////////////////SYSTEM INFO/////////////////////////////////////////////////////////////////////////////////////

	sSoftwareVersion					: STRING := ' 1.0 ';
	sSoftwareDate						: STRING := '03/06/2026';
	sTC3Version							: STRING := ' v3.1.4026.22, Runtime v3.1.4026.22 ';
	sHMIVersion							: STRING := ' 14.13';
	sSystemName							: STRING := 'LT-WH IPX8';
	sProjectID							: STRING := ' TE 11108' ;
	sAplication                     	: STRING ;
	sHMIServer                			: STRING := ' 14.13 ';
	
/////////////////////////////////////////////////////////////////////////////////////MANUAL/////////////////////////////////////////////////////////////////////////////////////

	bEnableManual						: BOOL;
	nMainRegion							: DINT;
	bManualModeOffFlag					: BOOL;
	bManualScreen						: BOOL;
	tonManualMode						: TON;
	bEnableSettings						: BOOL;
	
	stAnimations						: ST_Animations;
	
	bProcessCylinder_Up					: BOOL;
	bProcessCylinder_Down2				: BOOL;
	
	bProcessDoor_Up2					: BOOL;
	bProcessDoor_Down					: BOOL;
	
	bSlideNestRight						: BOOL;
	bSlideNestLeft						: BOOL;
	
	bLeaktester1_Start					: BOOL;
	bLeaktester2_Start					: BOOL;
	bLeaktester1_Stop					: BOOL;
	bLeaktester2_Stop					: BOOL;
	bLeaktester1_Reset					: BOOL;
	bLeaktester2_Reset					: BOOL;
	
	bProcessCylinderDownEnable			: BOOL;
	
	//Probes
	bSetTolerances						: BOOL;
	abPresetProbe						: ARRAY [1..8] OF BOOL;
	bSetCalibrationBlock1				: BOOL;
	bSetCalibrationBlock2				: BOOL;
	bEnableSetCablibrationBlock1		: BOOL;
	bEnableSetCablibrationBlock2		: BOOL;
	bSetDistances						: BOOL;
	
	
	
	
END_VAR

VAR_GLOBAL PERSISTENT
	
	stTimers							: ST_Timers;
	stStatisticsHMI						: ARRAY [0..5] OF ST_StatisticsHMI;	//0: Nest1
																	//1: Nest2
																	//2: Leak Tester 1
																	//3: Leak Tester 2
																	//4: Height Test 1
																	//5: Height Test 2
																	
														
	/////////////////////////////////////////////////////////////////////////////////////SETTINGS/////////////////////////////////////////////////////////////////////////////////////	
	
	//TwinSAFE
	
	nAirPressureMaxValue				: UINT;	
	nAirPressureMinValue				: UINT;	
	abMachineDefinition					: ARRAY[1..5] OF  BOOL;
	stTableCycleDataNest1				: ARRAY[0..2000] OF ST_TableCycleData;
	stTableCycleDataNest2				: ARRAY[0..2000] OF ST_TableCycleData;
	
	bNest1Flag							: BOOL;
	bNest2Flag							: BOOL;


	
END_VAR

// ---- GVLs/GVL_Master.TcGVL
VAR_GLOBAL
////////////////////////////////////////:	///////////////////////////////////////////////////
/////////////////////////////////////////////////////////////////////////////////////GENERIC/////////////////////////////////////////////////////////////////////////////////////

	// PowerUP 
	tonSystemPowerUP				:TON;
	tSystemPowerUP_Time				:TIME								:=T#3S;
	bSystemPoweringUP				:BOOL								:=TRUE; //Global System PowerUP Flag
	
	fbSystemShutDown     	        : NT_Shutdown;
	stButtonsLamps					: ST_ButtonsLamps;
	rtrigButton             		: ARRAY[1..3] OF Tc2_Standard.R_TRIG;
	ftrigButton             		: ARRAY[1..3] OF Tc2_Standard.F_TRIG; 
	stPuls							: ST_Puls;		

	stCycleDataNest1				: ST_CycleData;
	stCycleDataNest2				: ST_CycleData;
	
	bWriteNest1						: BOOL;
	bWriteNest2						: BOOL;
	bCSVDone						: BOOL;
	bCSVReady						: BOOL;
	bAutocycleIDLE					: BOOL;
	bDoorOpenedFlag					: BOOL;
	
	bRejectPartFault				: BOOL;
	bRejectPartOutTime				: BOOL;
	bCSVError						: BOOL;
	
	NetAmsIdLocal        	       	: T_AmsNetId;// := '172.18.236.164.1.1'; // AMS-ID for com port setup 
	bReadAMSNetID					: BOOL;
	fbGetLocalAMSNetID				: FB_GetLocalAmsNetId;
	
	fbGetDeviceNetId				: IOF_GetDeviceNetId;
	NetAmsIdDevice					: T_AmsNetId;
	
	bOpenDoorCycleFault				: BOOL;
	
	
	
/////////////////////////////////////////////////////////////////////////////////////Event Log/////////////////////////////////////////////////////////////////////////////////////
	
	stStationEvents				: ARRAY[0..4] OF  ST_StationEvents;//0: GENERAL
																	//1: Leak Test
																	//1: Height Test
																	//3: Vision Inspection
																	//4: Cylinders
	astActiveEvents				: ARRAY [0..50] OF ST_ActiveEvents;
	stEventsAssigment			: ST_EventsAssigmentGeneral;
	bMachineMessages			: BOOL;
	sMachineMessage				: STRING;

/////////////////////////////////////////////////////////////////////////////////////MACHINE CONTROL////////////////////////////////////////////////////////////////////////////
	
	stMachineStatus					: ST_MachineStatus;	
	stMasterCtrl					: ST_MasterCTRL;
	bStatisticsTest					: ARRAY[0..5] OF  BOOL;
	
	
////////////////////////////////////////////////////////////////////////////////////SYSTEM////////////////////////////////////////////////////////////////////////////

	stSystemTime				: TIMESTRUCT;
	sSystemTime					: STRING(255);
	sSystemDate					: STRING(255);

////////////////////////////////////////////////////////////////////////////////////SAFETY////////////////////////////////////////////////////////////////////////////

	bDoorClosingFlag				: BOOL;
	bDoorOpeningFlag				: BOOL;
	bProcessDoorClosedConditionFlag	: BOOL;
	tonSafety						: TON;
	bProcessCylinderSafetyPosition	: BOOL;
	bProcessDoorUpInitialising		: BOOL;
	
END_VAR

// ---- GVLs/GVL_Stations.TcGVL
VAR_GLOBAL

	stLeakTesters							: ST_LeakTester;	
	stHeightTests							: ST_HeightTest;
	stProcessCylinder						: ST_ProcessCylinder;
	stProcessDoor							: ST_ProcessDoor;
	stSlideNest								: ST_SlideNest;
	
END_VAR

// ---- POUs/A_MASTER/A_1_PRG_Main_Master.TcPOU
PROGRAM A_1_PRG_Main_Master
VAR
	
	
	fbStringFormatter       				: Tc2_Utilities.FB_FormatString;
	fbEventsManager							: FB_EventsManager;
	bResetEvents							: BOOL;
	
	ntShutdown								: TC2_Utilities.NT_Shutdown;
	closeChrome 							: NT_StartProcess;
	bCloseChromeBusy						: BOOL;
	tonCloseChromeBusy						: TON;
	//fbUserLog								: FB_UserLog;
	
	fbSystemTime							: NT_GetTime;
	
	fbScaleAirSupply						: FB_Scale;
	
	i										: DINT; //index quit HMI
	
	//Statistics
	rGoodStatistics							: ARRAY [0..1] OF R_TRIG;
	rBadStatistics							: ARRAY [0..1] OF R_TRIG;
	rEfficency								: STRING(510);


				
END_VAR

/////////////////////////////////////////////////////////////////////////////////////GENERAL/////////////////////////////////////////////////////////////////////////////////////
A_3_PRG_FaultHandling();
b_ACT_UserLogout();
a_ACT_ButtonsLamps();
d_ACT_ShutdownAndQuit();
f_ACT_TerminalInfo();
g_ACT_Manual();
h_ACT_Statistics();
i_ACT_TwinSAFE();

C_1_PRG_MainHMI();

PRG_Puls();

// System PowerUP CTRL
tonSystemPowerUP(IN:=bSystemPoweringUP, PT:=tSystemPowerUP_Time);
IF tonSystemPowerUP.Q THEN 
bSystemPoweringUP:=FALSE;
END_IF

/////////////////////////////////////////////////////////////////////////////////////STATIONS/////////////////////////////////////////////////////////////////////////////////////
	
	B_2_1_PRG_Master_Height_Test();	
	B_1_1_PRG_Master_Leak_Test();
	B_4_1_PRG_Master_ProcessCylinder();
	B_4_2_PRG_Master_ProcessDoor();
	B_4_3_PRG_Master_SlideNest();

/////////////////////////////////////////////////////////////////////////////////////PROCESS/////////////////////////////////////////////////////////////////////////////////////

A_2_PRG_MachineCtrl();

/////////////////////////////////////////////////////////////////////////////////////EVENT LOG/////////////////////////////////////////////////////////////////////////////////////

fbEventsManager	(			//INPUTS
							bPulse 							:= stPuls.bFlash10Hz, 
							bResetFaults 					:= dw_T04_EL1918.iResetButton, 
							stStationEvents 				:= stStationEvents,
							sSystemTime						:= sSystemTime,
							sSystemDate						:= sSystemDate,
 							stEventsAssigment				:= stEventsAssigment,
							bDataWritedInCSV				:= ,
							nArraySize						:= 5,
							bMachineMessage					:= sMachineMessage,
							
							//OUTPUTS
							astActiveEvents 				=> astActiveEvents,
							astEventsHistory				=> astEventsHistory,
							);



////////////////////////////////////////////////////////////////////////////////////SYSTEM DATE & TIME/////////////////////////////////////////////////////////////////////////////////////

fbSystemTime( START := stPuls.bFlash10Hz, TIMESTR => stSystemTime);
	

sSystemTime					:= 	CONCAT( STR1 := WORD_TO_STRING(stSystemTime.wHour), STR2 := CONCAT( STR1 := ':', STR2 := 
								CONCAT( STR1 := WORD_TO_STRING(stSystemTime.wMinute), STR2 := 
								CONCAT(STR1 := ':', STR2 := WORD_TO_STRING(stSystemTime.wSecond)))));
								
sSystemDate					:= 	CONCAT( STR1 := WORD_TO_STRING(stSystemTime.wDay), STR2 := 
								CONCAT(STR1 := '_', STR2 := CONCAT(STR1 := WORD_TO_STRING(stSystemTime.wMonth), STR2 := 
								CONCAT(STR1 := '_', STR2 := WORD_TO_STRING(stSystemTime.wYear)))));


stCycleDataNest1.nNest		:= 1;
stCycleDataNest2.nNest		:= 2;

////////////////////////////////////////////////////////////////////////////////////CSV////////////////////////////////////////////////////////////////////////////	

	

D_1_PRG_CycleDataCSV( 	stCycleDataNest1 	:= stCycleDataNest1,
						stCycleDataNest2 	:= stCycleDataNest2,
						bWriteNest1			:= bWriteNest1,
						bWriteNest2			:= bWriteNest2,
						bCSVDone			=> bCSVDone,
						bReady				=> bCSVReady);
	
fbGetLocalAMSNetID(
					bExecute	:= bReadAMSNetID,
					AddrString => NetAmsIdLocal);	

fbGetDeviceNetId(	START		:= 	bReadAMSNetID,
					DEVICEID	:= 3,
					DeviceNetId	=> 	NetAmsIdDevice);

ACTION a_ACT_ButtonsLamps:
//===================================================================
stButtonsLamps.bStartButtonFallingEdge 		:= ftrigButton[1].Q ;
stButtonsLamps.bStartButtonRisingEdge 		:= rtrigButton[1].Q ;
stButtonsLamps.bStopButtonFallingEdge 		:= ftrigButton[2].Q ; 
stButtonsLamps.bStopButtonRisingEdge 		:= rtrigButton[2].Q ;  
stButtonsLamps.bResetButtonFallingEdge 		:= ftrigButton[3].Q ;
stButtonsLamps.bResetButtonRisingEdge 		:= rtrigButton[3].Q ;



ftrigButton[1](CLK 							:= dw_T08_EL1809.iStartButoon);
rtrigButton[1](CLK							:= dw_T08_EL1809.iStartButoon);
ftrigButton[2](CLK							:= NOT dw_T08_EL1809.iStopButton);
rtrigButton[2](CLK							:= NOT dw_T08_EL1809.iStopButton);
ftrigButton[3](CLK							:= dw_T04_EL1918.iResetButton);
rtrigButton[3](CLK							:= dw_T04_EL1918.iResetButton);

dw_T09_EL2809.qResetButtonLED				:= (stMachineStatus.bFault AND stPuls.bFlash1Hz) OR (stMachineStatus.bStopped AND stPuls.bFlash2Hz) OR stMachineStatus.bManualMode;
dw_T09_EL2809.qStartButtonLED				:= (stMachineStatus.bReadyToStart AND stPuls.bFlash1Hz) OR stMachineStatus.bAutoCycle OR stMachineStatus.bManualMode;
END_ACTION

ACTION b_ACT_UserLogout:
tonHMIAliveOn(IN := bHMIAlive, PT:= T#2S);

tonHMIAliveOff(IN := NOT bHMIAlive, PT:= T#2S);

bOutHMI := tonHMIAliveOn.Q OR tonHMIAliveOff.Q;
END_ACTION

ACTION d_ACT_ShutdownAndQuit:
tonCloseChromeBusy( IN := bQuitHmi, PT := T#5S);
IF  tonCloseChromeBusy.Q THEN
	
	bQuitHmi			:= FALSE;

END_IF

closeChrome(
    NetId := NetAmsIdLocal,
    PathStr := 'C:\Windows\System32\mshta vbscript:Execute("CreateObject(""WScript.Shell"").Run ""powershell -c',
    DirName := 'C:\Windows\System32\WindowsPowerShell\v1.0',
    ComndLine := 'taskkill /F /IM msedge.exe /T"", 0: window.close")',
    Start := bQuitHmi,
    TmOut := DEFAULT_ADS_TIMEOUT,
	BUSY => bCloseChromeBusy
);


ntShutdown(NETID := NetAmsIdLocal, DELAY := 5, START := bShutDown);

IF dw_T08_EL1809.iStartButoon THEN
	IF ftrigButton[2].Q THEN
		i:= i+1;
	END_IF
	IF i>=3 THEN;
		bQuitHmi:=TRUE;
	END_IF
ELSE
	i:=0;
END_IF
END_ACTION

ACTION f_ACT_TerminalInfo:
dw_T01_EK1100.stTerminalInfo.fbTerminalInfo( 	nTerminalState						:= dw_T01_EK1100.stTerminalInfo.nTerminal_State,
												sTerminalState						=> dw_T01_EK1100.stTerminalInfo.sTerminalInfo,
												bTerminalOperational				=> dw_T01_EK1100.stTerminalInfo.bTerminalOperational);
									
dw_T02_EL6070.stTerminalInfo.fbTerminalInfo( 	nTerminalState						:= dw_T02_EL6070.stTerminalInfo.nTerminal_State,
												sTerminalState						=> dw_T02_EL6070.stTerminalInfo.sTerminalInfo,
												bTerminalOperational				=> dw_T02_EL6070.stTerminalInfo.bTerminalOperational);

dw_T03_EL6910.stTerminalInfo.fbTerminalInfo( 	nTerminalState						:= dw_T03_EL6910.stTerminalInfo.nTerminal_State,
												sTerminalState						=> dw_T03_EL6910.stTerminalInfo.sTerminalInfo,
												bTerminalOperational				=> dw_T03_EL6910.stTerminalInfo.bTerminalOperational);
												
dw_T04_EL1918.stTerminalInfo.fbTerminalInfo(	nTerminalState						:= dw_T04_EL1918.stTerminalInfo.nTerminal_State,
												sTerminalState						=> dw_T04_EL1918.stTerminalInfo.sTerminalInfo,
												bTerminalOperational				=> dw_T04_EL1918.stTerminalInfo.bTerminalOperational);
												
dw_T05_EL1918.stTerminalInfo.fbTerminalInfo(	nTerminalState						:= dw_T05_EL1918.stTerminalInfo.nTerminal_State,
												sTerminalState						=> dw_T05_EL1918.stTerminalInfo.sTerminalInfo,
												bTerminalOperational				=> dw_T05_EL1918.stTerminalInfo.bTerminalOperational);
												
dw_T06_EL2904.stTerminalInfo.fbTerminalInfo(	nTerminalState						:= dw_T06_EL2904.stTerminalInfo.nTerminal_State,
												sTerminalState						=> dw_T06_EL2904.stTerminalInfo.sTerminalInfo,
												bTerminalOperational				=> dw_T06_EL2904.stTerminalInfo.bTerminalOperational);
												
dw_T07_EL9410.stTerminalInfo.fbTerminalInfo(	nTerminalState						:= dw_T07_EL9410.stTerminalInfo.nTerminal_State,
												sTerminalState						=> dw_T07_EL9410.stTerminalInfo.sTerminalInfo,
												bTerminalOperational				=> dw_T07_EL9410.stTerminalInfo.bTerminalOperational);
											
dw_T08_EL1809.stTerminalInfo.fbTerminalInfo(	nTerminalState						:= dw_T08_EL1809.stTerminalInfo.nTerminal_State,
												sTerminalState						=> dw_T08_EL1809.stTerminalInfo.sTerminalInfo,
												bTerminalOperational				=> dw_T08_EL1809.stTerminalInfo.bTerminalOperational);
												
dw_T09_EL2809.stTerminalInfo.fbTerminalInfo(	nTerminalState						:= dw_T09_EL2809.stTerminalInfo.nTerminal_State,
												sTerminalState						=> dw_T09_EL2809.stTerminalInfo.sTerminalInfo,
												bTerminalOperational				=> dw_T09_EL2809.stTerminalInfo.bTerminalOperational);
												
												
dw_T10_EL3058.stTerminalInfo.fbTerminalInfo(	nTerminalState						:= dw_T10_EL3058.stTerminalInfo.nTerminal_State,
												sTerminalState						=> dw_T10_EL3058.stTerminalInfo.sTerminalInfo,
												bTerminalOperational				=> dw_T10_EL3058.stTerminalInfo.bTerminalOperational);
												
dw_T11_EL1918.stTerminalInfo.fbTerminalInfo(	nTerminalState						:= dw_T11_EL1918.stTerminalInfo.nTerminal_State,
												sTerminalState						=> dw_T11_EL1918.stTerminalInfo.sTerminalInfo,
												bTerminalOperational				=> dw_T11_EL1918.stTerminalInfo.bTerminalOperational);
												
dw_T12_EL6633.stTerminalInfo.fbTerminalInfo(	nTerminalState						:= dw_T12_EL6633.stTerminalInfo.nTerminal_State,
												sTerminalState						=> dw_T12_EL6633.stTerminalInfo.sTerminalInfo,
												bTerminalOperational				=> dw_T12_EL6633.stTerminalInfo.bTerminalOperational);
												
//add boxes

Probes.stTerminalInfo.fbTerminalInfo(			nTerminalState						:= Probes.stTerminalInfo.nTerminal_State,
												sTerminalState						=> Probes.stTerminalInfo.sTerminalInfo,
												bTerminalOperational				=> Probes.stTerminalInfo.bTerminalOperational);
END_ACTION

ACTION g_ACT_Manual:
tonManualMode( IN := bManualScreen, PT := T#100MS);

IF stMachineStatus.bReadyToStart THEN
	bEnableManual											:= TRUE;
ELSE bEnableManual											:= FALSE;
END_IF
	
bManualModeOffFlag										:= FALSE;



IF bManualScreen  THEN
	
	stMasterCtrl.bManualModeRequest							:= TRUE;
	
	IF (stMachineStatus.eMachineState <> E_MachineState.MANUAL_MODE) AND tonManualMode.Q THEN
				
		stMasterCtrl.bManualModeRequest							:= FALSE; 
		bManualModeOffFlag										:= TRUE;
		
	END_IF
	
ELSE 
	stMasterCtrl.bManualModeRequest							:= FALSE; 
												
END_IF
END_ACTION

ACTION h_ACT_Statistics:

stStatisticsHMI[0].sName			:= 'TEST ZONE - LH';
stStatisticsHMI[1].sName			:= 'TEST ZONE - RH';



rGoodStatistics[0]( CLK := stCycleDataNest1.bPass);
rBadStatistics[0]( CLK := stCycleDataNest1.bFail);
rGoodStatistics[1]( CLK := stCycleDataNest2.bPass);
rBadStatistics[1]( CLK := stCycleDataNest2.bFail);

IF 	rGoodStatistics[0].Q  THEN
	
	stStatisticsHMI[0].nGood		:= stStatisticsHMI[0].nGood + 1;

ELSIF 	rBadStatistics[0].Q  THEN
	
	stStatisticsHMI[0].nBad			:= stStatisticsHMI[0].nBad + 1;
		
END_IF
								


IF stStatisticsHMI[0].bResetGood THEN
	stStatisticsHMI[0].nGood		:= 0;
END_IF

IF stStatisticsHMI[0].bResetBad THEN
	stStatisticsHMI[0].nBad			:= 0;
END_IF



IF 	rGoodStatistics[1].Q  THEN
	
	stStatisticsHMI[1].nGood		:= stStatisticsHMI[1].nGood + 1;

ELSIF 	rBadStatistics[1].Q  THEN
	
	stStatisticsHMI[1].nBad			:= stStatisticsHMI[1].nBad + 1;
		
END_IF
								


IF stStatisticsHMI[1].bResetGood THEN
	stStatisticsHMI[1].nGood		:= 0;
END_IF

IF stStatisticsHMI[1].bResetBad THEN
	stStatisticsHMI[1].nBad			:= 0;
END_IF



IF (( stStatisticsHMI[0].nGood + stStatisticsHMI[0].nBad) <> 0) THEN
	
	rEfficency							:= LREAL_TO_FMTSTR(in := (DINT_TO_REAL(stStatisticsHMI[0].nGood) /( DINT_TO_REAL(stStatisticsHMI[0].nGood) + DINT_TO_REAL(stStatisticsHMI[0].nBad))) * 100.0,iPrecision := 2, bRound := TRUE);
	stStatisticsHMI[0].nEfficency		:= CONCAT(STR1 := '%', STR2 := (rEfficency));

ELSE stStatisticsHMI[0].nEfficency		:= CONCAT(STR1 := '%', STR2 := (DINT_TO_STRING(0)));
	
END_IF

IF (( stStatisticsHMI[1].nGood + stStatisticsHMI[1].nBad) <> 0) THEN
	
	rEfficency							:= LREAL_TO_FMTSTR(in := (DINT_TO_REAL(stStatisticsHMI[1].nGood) /( DINT_TO_REAL(stStatisticsHMI[1].nGood) + DINT_TO_REAL(stStatisticsHMI[1].nBad))) * 100.0,iPrecision := 2, bRound := TRUE);
	stStatisticsHMI[1].nEfficency		:= CONCAT(STR1 := '%', STR2 := (rEfficency));

ELSE stStatisticsHMI[1].nEfficency		:= CONCAT(STR1 := '%', STR2 := (DINT_TO_STRING(0)));
	
END_IF
END_ACTION

ACTION i_ACT_TwinSAFE:
	
stTwinSAFE.iSafetyErrorAcknowledge		:= dw_T04_EL1918.iResetButton;

fbScaleAirSupply( 			nRawValue						:= UINT_TO_REAL(GVL_IO.dw_T10_EL3058.iMainPressure),
							X1								:= 0,
							X2								:= 32768,
							Y1								:= 0,
							Y2								:= 10,
							
							nOutPut							=> stTwinSAFE.iAirSupplyMeasurement);

stTwinSAFE.iAirPressureMaxValue			:= nAirPressureMaxValue;
stTwinSAFE.iAirPressureMinValue			:= nAirPressureMinValue;
stTwinSAFE.iProcessDoorClosing			:= bDoorClosingFlag;
					

////////////////////////////////////////////////////////////TwinSAFE Outputs reading//////////////////////////////////////////////////////////

dw_T06_EL2904.qEnableAirSupply_PSR1								:= SEL((dw_T06_EL2904_Reading.bResult[1]=1),FALSE,TRUE);
dw_T06_EL2904.qResetAirSupply_PSR2								:= SEL((dw_T06_EL2904_Reading.bResult[2]=1),FALSE,TRUE);
dw_T06_EL2904.qLockMainDoor										:= SEL((dw_T06_EL2904_Reading.bResult[3]=1),FALSE,TRUE);
dw_T06_EL2904.qLockProcessCylinder								:= SEL((dw_T06_EL2904_Reading.bResult[4]=1),FALSE,TRUE);

dw_T06_EL2904_Reading.fbReadOutSafety06[1]( 	sNetId 			:=NetAmsIdDevice,
	                					 		nSlaveAddr 		:=1006,
					 							nSubIndex 		:=0001,
					 							nIndex 			:=16#7001 ,
					 							pDstBuf 		:=ADR(dw_T06_EL2904_Reading.bResult[1]),
					 							cbBufLen 		:=SIZEOF(dw_T06_EL2904_Reading.bResult[1]),
					 							bExecute 		:= stPuls.bFlash4Hz,
					 							tTimeout 		:= T#500MS,
					 							bBusy 			=> dw_T06_EL2904_Reading.bBusy[1],
					 							bError 			=> dw_T06_EL2904_Reading.berror[1]);
												
dw_T06_EL2904_Reading.fbReadOutSafety06[2]( 	sNetId 			:= NetAmsIdDevice,
	                					 		nSlaveAddr 		:=1006,
					 							nSubIndex 		:=0002,
					 							nIndex 			:=16#7001 ,
					 							pDstBuf 		:=ADR(dw_T06_EL2904_Reading.bResult[2]),
					 							cbBufLen 		:=SIZEOF(dw_T06_EL2904_Reading.bResult[2]),
					 							bExecute 		:= stPuls.bFlash4Hz,
					 							tTimeout 		:= T#500MS,
					 							bBusy 			=> dw_T06_EL2904_Reading.bBusy[2],
					 							bError 			=> dw_T06_EL2904_Reading.berror[2]);
												
dw_T06_EL2904_Reading.fbReadOutSafety06[3]( 	sNetId 			:=NetAmsIdDevice,
	                					 		nSlaveAddr 		:=1006,
					 							nSubIndex 		:=0003,
					 							nIndex 			:=16#7001 ,
					 							pDstBuf 		:=ADR(dw_T06_EL2904_Reading.bResult[3]),
					 							cbBufLen 		:=SIZEOF(dw_T06_EL2904_Reading.bResult[3]),
					 							bExecute 		:= stPuls.bFlash4Hz,
					 							tTimeout 		:= T#500MS,
					 							bBusy 			=> dw_T06_EL2904_Reading.bBusy[3],
					 							bError 			=> dw_T06_EL2904_Reading.berror[3]);
											
dw_T06_EL2904_Reading.fbReadOutSafety06[4]( 	sNetId 			:= NetAmsIdDevice,
	                					 		nSlaveAddr 		:=1006,
					 							nSubIndex 		:=0004,
					 							nIndex 			:=16#7001 ,
					 							pDstBuf 		:=ADR(dw_T06_EL2904_Reading.bResult[4]),
					 							cbBufLen 		:=SIZEOF(dw_T06_EL2904_Reading.bResult[4]),
					 							bExecute 		:= stPuls.bFlash4Hz,
					 							tTimeout 		:= T#500MS,
					 							bBusy 			=> dw_T06_EL2904_Reading.bBusy[4],
					 							bError 			=> dw_T06_EL2904_Reading.berror[4]);
END_ACTION

END_PROGRAM

// ---- POUs/A_MASTER/A_3_PRG_FaultHandling.TcPOU
PROGRAM A_3_PRG_FaultHandling
VAR
	

	bEventsFlag					: ARRAY [0..100] OF BOOL;
	i							: DINT;
	Counter						: CTU;			



END_VAR

a_ACT_Set_Events();
/////////////////////////////////////////////////////////////////////////////////////MASTER FAULT MONITORS////////////////////////////////////////////////////////////////////////////////////


stMasterCtrl.bNoFault 												:= 	NOT stStationEvents[0].bFault AND NOT stStationEvents[1].bFault AND
                                            							NOT stStationEvents[2].bFault AND NOT stStationEvents[3].bFault AND NOT stStationEvents[4].bFault
																		AND NOT stStationEvents[5].bFault;

stMasterCtrl.bCycleStopRequest										:= stStationEvents[0].bCycleStopRequest OR stStationEvents[1].bCycleStopRequest OR
																		stStationEvents[2].bCycleStopRequest OR stStationEvents[3].bCycleStopRequest OR stStationEvents[4].bCycleStopRequest
																		OR stStationEvents[5].bCycleStopRequest;

ACTION a_ACT_Set_Events:
/////////////////////////////////////////////////////////////////////////////////////TwinSAFE/////////////////////////////////////////////////////////////////////////////////////

stStationEvents[0].aEvents[0].bFault						:= TRUE;
stStationEvents[0].aEvents[0].bEventFlag					:= stTwinSAFE.qAirErrorSignal;
stStationEvents[0].aEvents[0].bEventText					:= 'Pressure Error';
stStationEvents[0].aEvents[0].sSolution						:= 'Check Air Supply system';

stStationEvents[0].aEvents[1].bFault						:= TRUE;
stStationEvents[0].aEvents[1].bEventFlag					:= stTwinSAFE.qAirPressureAbove;
stStationEvents[0].aEvents[1].bEventText					:= 'System overpressurized' ;
stStationEvents[0].aEvents[1].sSolution						:= 'set the main valve to the right pressure';

stStationEvents[0].aEvents[2].bFault						:= TRUE;
stStationEvents[0].aEvents[2].bEventFlag					:= stTwinSAFE.qAirPressureBelow;
stStationEvents[0].aEvents[2].bEventText					:= 'Not enough pressure in the system' ;
stStationEvents[0].aEvents[2].sSolution						:= 'set the main valve to the right pressure and check the air supply';

stStationEvents[0].aEvents[3].bFault						:= TRUE;
stStationEvents[0].aEvents[3].bEventFlag					:= NOT dw_T04_EL1918.iEStopChannel1 AND dw_T04_EL1918.iEStopChannel2;
stStationEvents[0].aEvents[3].bEventText					:= 'E-STOP CH1 malfunction' ;
stStationEvents[0].aEvents[3].sSolution						:= 'Check E-STOP CH1';

stStationEvents[0].aEvents[4].bFault						:= TRUE;
stStationEvents[0].aEvents[4].bEventFlag					:= dw_T04_EL1918.iEStopChannel1 AND NOT dw_T04_EL1918.iEStopChannel2;
stStationEvents[0].aEvents[4].bEventText					:= 'E-STOP CH2 malfunction' ;
stStationEvents[0].aEvents[4].sSolution						:= 'Check E-STOP CH2';

stStationEvents[0].aEvents[5].bFault						:= TRUE;
stStationEvents[0].aEvents[5].bEventFlag					:= stTwinSAFE.qE_StopPressed;
stStationEvents[0].aEvents[5].bEventText					:= 'E-STOP Pressed' ;
stStationEvents[0].aEvents[5].sSolution						:= 'Release E-STOP';

stStationEvents[0].aEvents[6].bFault						:= TRUE;
stStationEvents[0].aEvents[6].bEventFlag					:= stTwinSAFE.qSafetyOk AND NOT stTwinSAFE.qSystemSafe;
stStationEvents[0].aEvents[6].bEventText					:= 'Safe system error' ;
stStationEvents[0].aEvents[6].sSolution						:= 'Check safety elements';

stStationEvents[0].aEvents[7].bFault						:= TRUE;
stStationEvents[0].aEvents[7].bEventFlag					:= NOT dw_T08_EL1809.iUP_OK;
stStationEvents[0].aEvents[7].bEventText					:= 'UP (Primary Power Supply) Stop Working' ;
stStationEvents[0].aEvents[7].sSolution						:= 'Check UP Power Supply';

stStationEvents[0].aEvents[8].bFault						:= TRUE;
stStationEvents[0].aEvents[8].bEventFlag					:= stTwinSAFE.qProcessDoorUnSafe;
stStationEvents[0].aEvents[8].bEventText					:= 'Process door movement unsafe' ;
stStationEvents[0].aEvents[8].sSolution						:= 'Reset system';

stStationEvents[0].aEvents[9].bFault						:= TRUE;
stStationEvents[0].aEvents[9].bEventFlag					:= stTwinSAFE.qTwoHandsUnsafe;
stStationEvents[0].aEvents[9].bEventText					:= 'Hands in unsafe position' ;
stStationEvents[0].aEvents[9].sSolution						:= 'Reset system';

stStationEvents[0].aEvents[10].bFault						:= TRUE;
stStationEvents[0].aEvents[10].bEventFlag					:= stTwinSAFE.qProcessCylinderUnsafe AND stTwinSAFE.qSafetyOk;
stStationEvents[0].aEvents[10].bEventText					:= 'Process cylinder Unsafe' ;
stStationEvents[0].aEvents[10].sSolution					:= 'Reset system';

stStationEvents[0].aEvents[11].bFault						:= TRUE;
stStationEvents[0].aEvents[11].bEventFlag					:= stTwinSAFE.qMainDoorUnsafe AND stTwinSAFE.qSafetyOk;
stStationEvents[0].aEvents[11].bEventText					:= 'Main Door Unsafe' ;
stStationEvents[0].aEvents[11].sSolution					:= 'Reset system';

stStationEvents[0].aEvents[12].bFault						:= TRUE;
stStationEvents[0].aEvents[12].bEventFlag					:= NOT dw_T08_EL1809.iUS_OK;
stStationEvents[0].aEvents[12].bEventText					:= 'US (Secondary Power Supply) Stop Working' ;
stStationEvents[0].aEvents[12].sSolution					:= 'Check US Power Supply';

stStationEvents[0].aEvents[13].bFault						:= TRUE;
stStationEvents[0].aEvents[13].bEventFlag					:= stTwinSAFE.qMainDoorUnsafe;
stStationEvents[0].aEvents[13].bEventText					:= 'Main door Unsafe' ;
stStationEvents[0].aEvents[13].sSolution					:= 'Close door and Reset system';

stStationEvents[0].aEvents[14].bFault						:= TRUE;
stStationEvents[0].aEvents[14].bEventTimer( IN := NOT stTwinSAFE.qSafetyOk AND (stMachineStatus.eMachineState = E_MachineState.SAFETY), PT := T#20S);
stStationEvents[0].aEvents[14].bEventFlag					:= stStationEvents[0].aEvents[14].bEventTimer.Q;
stStationEvents[0].aEvents[14].bEventText					:= 'Safe system init timeout' ;
stStationEvents[0].aEvents[14].sSolution					:= 'Check safety components, reset system';

stStationEvents[0].aEvents[15].bFault						:= TRUE;
stStationEvents[0].aEvents[15].bEventTimer(IN := stTwinSAFE.qComError OR stTwinSAFE.qFBError OR stTwinSAFE.qOtherError, PT := T#1S);
stStationEvents[0].aEvents[15].bEventFlag					:= stStationEvents[0].aEvents[15].bEventTimer.Q;
stStationEvents[0].aEvents[15].bEventText					:= 'Safety System error' ;
stStationEvents[0].aEvents[15].sSolution					:= 'Close door and Reset system';

stStationEvents[0].aEvents[16].bFault						:= TRUE;
stStationEvents[0].aEvents[16].bEventFlag					:= bRejectPartFault;
stStationEvents[0].aEvents[16].bEventText					:= 'Wrong part taken andput in the reject chute' ;
stStationEvents[0].aEvents[16].sSolution					:= 'Put parts in reject shutter and restart system';


stStationEvents[0].aEvents[18].bCycleStopRequest			:= TRUE;
stStationEvents[0].aEvents[18].bEventTimer(IN := dw_T08_EL1809.iRejectSensor, PT := T#3S);
stStationEvents[0].aEvents[18].bEventFlag					:= stStationEvents[0].aEvents[18].bEventTimer.Q;
stStationEvents[0].aEvents[18].bEventText					:= 'Reject chute full' ;
stStationEvents[0].aEvents[18].sSolution					:= 'Empty reject chute';

stStationEvents[0].aEvents[19].bFault						:= TRUE;
stStationEvents[0].aEvents[19].bEventTimer(IN := NOT dw_T08_EL1809.iStopButton, PT := T#3S);
stStationEvents[0].aEvents[19].bEventFlag					:= stStationEvents[0].aEvents[19].bEventTimer.Q;
stStationEvents[0].aEvents[19].bEventText					:= 'Immediate Stop requested' ;
stStationEvents[0].aEvents[19].sSolution					:= '';





/////////////////////////////////////////////////////////////////////////////////////Cards status/////////////////////////////////////////////////////////////////////////////////////

stStationEvents[0].aEvents[20].bFault						:= TRUE;
stStationEvents[0].aEvents[20].bEventFlag					:= NOT stMachineStatus.bSystemPowerUp AND dw_T01_EK1100.stTerminalInfo.nTerminal_State <> 8;
stStationEvents[0].aEvents[20].bEventText					:= 'T01_EK1100 card in fault' ;
stStationEvents[0].aEvents[20].sSolution					:= 'Reset System';

stStationEvents[0].aEvents[21].bFault						:= TRUE;
stStationEvents[0].aEvents[21].bEventFlag					:= NOT stMachineStatus.bSystemPowerUp AND dw_T02_EL6070.stTerminalInfo.nTerminal_State <> 8;
stStationEvents[0].aEvents[21].bEventText					:= 'T02_EL6070 card in fault' ;
stStationEvents[0].aEvents[21].sSolution					:= 'Reset System';

stStationEvents[0].aEvents[22].bFault						:= TRUE;
stStationEvents[0].aEvents[22].bEventFlag					:= NOT stMachineStatus.bSystemPowerUp AND dw_T03_EL6910.stTerminalInfo.nTerminal_State <> 8;
stStationEvents[0].aEvents[22].bEventText					:= 'T03_EL6910 card in fault' ;
stStationEvents[0].aEvents[22].sSolution					:= 'Reset System';

stStationEvents[0].aEvents[23].bFault						:= TRUE;
stStationEvents[0].aEvents[23].bEventFlag					:= NOT stMachineStatus.bSystemPowerUp AND dw_T04_EL1918.stTerminalInfo.nTerminal_State <> 8;
stStationEvents[0].aEvents[23].bEventText					:= 'T04_EL1918 card in fault' ;
stStationEvents[0].aEvents[23].sSolution					:= 'Reset System';

stStationEvents[0].aEvents[24].bFault						:= TRUE;
stStationEvents[0].aEvents[24].bEventFlag					:= NOT stMachineStatus.bSystemPowerUp AND dw_T05_EL1918.stTerminalInfo.nTerminal_State <> 8;
stStationEvents[0].aEvents[24].bEventText					:= 'T05_EL1918 card in fault' ;
stStationEvents[0].aEvents[24].sSolution					:= 'Reset System';

stStationEvents[0].aEvents[25].bFault						:= TRUE;
stStationEvents[0].aEvents[25].bEventFlag					:= NOT stMachineStatus.bSystemPowerUp AND dw_T06_EL2904.stTerminalInfo.nTerminal_State <> 8;
stStationEvents[0].aEvents[25].bEventText					:= 'T06_EL2904 card in fault' ;
stStationEvents[0].aEvents[25].sSolution					:= 'Reset System';

stStationEvents[0].aEvents[26].bFault						:= TRUE;
stStationEvents[0].aEvents[26].bEventFlag					:= NOT stMachineStatus.bSystemPowerUp AND dw_T07_EL9410.stTerminalInfo.nTerminal_State <> 8;
stStationEvents[0].aEvents[26].bEventText					:= 'T07_EL9410 card in fault' ;
stStationEvents[0].aEvents[26].sSolution					:= 'Reset System';

stStationEvents[0].aEvents[27].bFault						:= TRUE;
stStationEvents[0].aEvents[27].bEventFlag					:= NOT stMachineStatus.bSystemPowerUp AND dw_T08_EL1809.stTerminalInfo.nTerminal_State <> 8;
stStationEvents[0].aEvents[27].bEventText					:= 'T08_EL1809 card in fault' ;
stStationEvents[0].aEvents[27].sSolution					:= 'Reset System';

stStationEvents[0].aEvents[28].bFault						:= TRUE;
stStationEvents[0].aEvents[28].bEventFlag					:= NOT stMachineStatus.bSystemPowerUp AND dw_T09_EL2809.stTerminalInfo.nTerminal_State <> 8;
stStationEvents[0].aEvents[28].bEventText					:= 'T09_EL2809 card in fault' ;
stStationEvents[0].aEvents[28].sSolution					:= 'Reset System';

stStationEvents[0].aEvents[29].bFault						:= TRUE;
stStationEvents[0].aEvents[29].bEventFlag					:= NOT stMachineStatus.bSystemPowerUp AND dw_T10_EL3058.stTerminalInfo.nTerminal_State <> 8;
stStationEvents[0].aEvents[29].bEventText					:= 'T10_EL3058 card in fault' ;
stStationEvents[0].aEvents[29].sSolution					:= 'Reset System';

stStationEvents[0].aEvents[30].bFault						:= TRUE;
stStationEvents[0].aEvents[30].bEventFlag					:= NOT stMachineStatus.bSystemPowerUp AND dw_T11_EL1918.stTerminalInfo.nTerminal_State <> 8;
stStationEvents[0].aEvents[30].bEventText					:= 'T11_EL1918 card in fault' ;
stStationEvents[0].aEvents[30].sSolution					:= 'Reset System';

stStationEvents[0].aEvents[31].bFault						:= TRUE;
stStationEvents[0].aEvents[31].bEventFlag					:= NOT stMachineStatus.bSystemPowerUp AND dw_T12_EL6633.stTerminalInfo.nTerminal_State <> 8 AND NOT abMachineDefinition[2];
stStationEvents[0].aEvents[31].bEventText					:= 'T12_EL6633 card in fault' ;
stStationEvents[0].aEvents[31].sSolution					:= 'Reset System';

//GENERAL
stStationEvents[0].aEvents[32].bFault						:= TRUE;
stStationEvents[0].aEvents[32].bEventFlag					:= bDoorClosingFlag AND (NOT dw_T05_EL1918.iLeftTouchButtonNO OR NOT dw_T05_EL1918.iRightTouchButtonNO);
stStationEvents[0].aEvents[32].bEventText					:= 'Hands out before door was closed' ;
stStationEvents[0].aEvents[32].sSolution					:= 'Reset System';

stStationEvents[0].aEvents[33].bFault						:= TRUE;
stStationEvents[0].aEvents[33].bEventFlag					:= ((stMachineStatus.eMachineState = E_MachineState.MANUAL_MODE) OR (stMachineStatus.eMachineState = E_MachineState.SYSTEM_AUTO_CYCLE ))
																AND bOutHMI;
stStationEvents[0].aEvents[33].bEventText					:= 'Out HMI while Machine was in Autocycle' ;
stStationEvents[0].aEvents[33].sSolution					:= 'Reset System';


stStationEvents[0].aEvents[34].bFault						:= TRUE;
stStationEvents[0].aEvents[34].bEventTimer(IN := (stMachineStatus.eMachineState = E_MachineState.SYSTEM_AUTO_CYCLE) AND NOT bAutocycleIDLE, PT := stTimers.tAutoCycleTimeOut );
stStationEvents[0].aEvents[34].bEventFlag					:= stStationEvents[0].aEvents[34].bEventTimer.Q;
stStationEvents[0].aEvents[34].bEventText					:= 'Auto Cycle Timeout' ;
stStationEvents[0].aEvents[34].sSolution					:= 'Reset System';

// PUCK LOCKER //Renan Added 06Jul26
stStationEvents[0].aEvents[35].bFault 						:= TRUE;
stStationEvents[0].aEvents[35].bEventFlag 					:= GVL_Stations.stPuckLocker.bUnexpectedRemovalFault;
stStationEvents[0].aEvents[35].bEventText 					:= 'Puck removed while locker pin was engaged';
stStationEvents[0].aEvents[35].sSolution 					:= 'Return puck to the locker position and acknowledge the alarm with Administrator access';



//STOP REQUEST

stStationEvents[0].aEvents[40].bCycleStopRequest			:= TRUE;
stStationEvents[0].aEvents[40].bEventFlag					:=  bOutHMI;
stStationEvents[0].aEvents[40].bEventText					:= 'Out HMI or User not logged in' ;
stStationEvents[0].aEvents[40].sSolution					:= '';

stStationEvents[0].aEvents[41].bCycleStopRequest			:= TRUE;
stStationEvents[0].aEvents[41].bEventTimer(IN := bAutocycleIDLE, PT := stTimers.tAutoCycleIDLETimeOut);
stStationEvents[0].aEvents[41].bEventFlag					:= stStationEvents[0].aEvents[41].bEventTimer.Q;
stStationEvents[0].aEvents[41].bEventText					:= 'Autocycle in IDLE Timeout' ;
stStationEvents[0].aEvents[41].sSolution					:= '';

stStationEvents[0].aEvents[42].bCycleStopRequest			:= TRUE;
stStationEvents[0].aEvents[42].bEventFlag					:= NOT dw_T08_EL1809.iStopButton;
stStationEvents[0].aEvents[42].bEventText					:= 'Stop Button Pressed' ;
stStationEvents[0].aEvents[42].sSolution					:= '';

stStationEvents[0].aEvents[43].bCycleStopRequest			:= TRUE;
stStationEvents[0].aEvents[43].bEventFlag					:=  stTwinSAFE.qMainDoorOpenned;
stStationEvents[0].aEvents[43].bEventText					:= 'Door openned ' ;
stStationEvents[0].aEvents[43].sSolution					:= 'Close door and Reset system to intilisation';


stStationEvents[0].aEvents[44].bCycleStopRequest			:= TRUE;
stStationEvents[0].aEvents[44].bEventFlag					:=  (stMachineStatus.eMachineState = E_MachineState.SYSTEM_AUTO_CYCLE) AND NOT bNest1Flag AND NOT bNest2Flag;
stStationEvents[0].aEvents[44].bEventText					:= 'No Nest enabled' ;
stStationEvents[0].aEvents[44].sSolution					:= 'Enable at least one Nest';


//MESSAGES

stStationEvents[0].aEvents[60].bMessage						:= TRUE;
stStationEvents[0].aEvents[60].bEventFlag					:=  bCSVError;
stStationEvents[0].aEvents[60].bEventText					:= 'CSV Not written ' ;
stStationEvents[0].aEvents[60].sSolution					:= '';
END_ACTION

END_PROGRAM

// ---- POUs/C_HMI/C_1_PRG_MainHMI.TcPOU
PROGRAM C_1_PRG_MainHMI
VAR
	
	bResetTest				: BOOL;
	i						: DINT;
	n						: DINT;//TABLE INDEX

END_VAR

a_ACT_MachineStatusBaner();
b_ACT_Timers();
c_ACT_IO();

bEnableSettings				:= (stMachineStatus.eMachineState = E_MachineState.STOPPED);
bOpenRejectDialog			:= bRejectPartDialog[0] OR bRejectPartDialog[1] OR bRejectPartDialog[2];
bProcessCylinderDownEnable	:= dw_T08_EL1809.iPartPresentNest1 AND dw_T08_EL1809.iPartPresentNest2 AND dw_T05_EL1918.iProcessDoorFB;

ACTION a_ACT_MachineStatusBaner:
//Machine status banner action
//SYSTEM POWER UP
IF stMachineStatus.bSystemPowerUp THEN	
	stStatusBanner.sMachineStatusText 							:= 'SYSTEM POWER UP';	
	stStatusBanner.nMachineStatusColour 						:= nWHITE;
	stStatusBanner.nMachineStatusTxtCol 						:= nBLACK;
	stStatusBanner.sBannerBckColor 								:= sWHITE;
	stStatusBanner.sBannerTextColor 							:= sBLACK;
END_IF

(* SYSTEM INITIALISING *)
IF stMachineStatus.bInitialising THEN	
	stStatusBanner.sMachineStatusText 							:= 'SYSTEM INITIALIZING';		
	stStatusBanner.nMachineStatusColour 						:= nYELLOW;
	stStatusBanner.nMachineStatusTxtCol 						:= nBLACK;
	stStatusBanner.sBannerBckColor 								:= sYELLOW;
	stStatusBanner.sBannerTextColor 							:= sBLACK;
END_IF

(* SAFETY *)
IF stMachineStatus.bSafety THEN	
	stStatusBanner.sMachineStatusText 							:= 'SYSTEM INITIALIZING';		
	stStatusBanner.nMachineStatusColour 						:= nYELLOW;
	stStatusBanner.nMachineStatusTxtCol 						:= nBLACK;
	stStatusBanner.sBannerBckColor 								:= sYELLOW;
	stStatusBanner.sBannerTextColor 							:= sBLACK;
END_IF


(* SYSTEM READY TO START FLASH ON *)
IF stMachineStatus.bReadyToStart AND stPuls.bFlash1Hz THEN
	stStatusBanner.sMachineStatusText 							:= 'SYSTEM READY TO START';		
	stStatusBanner.nMachineStatusColour 						:= nGREEN;
	stStatusBanner.nMachineStatusTxtCol 						:= nWHITE;
	stStatusBanner.sBannerBckColor 								:= sGREEN;
	stStatusBanner.sBannerTextColor 							:= sWHITE;
ELSIF stMachineStatus.bReadyToStart AND NOT stPuls.bFlash1Hz THEN	
	stStatusBanner.sMachineStatusText 							:= 'SYSTEM READY TO START';		
	stStatusBanner.nMachineStatusColour 						:= nWHITE;
	stStatusBanner.nMachineStatusTxtCol 						:= nGREEN;
	stStatusBanner.sBannerBckColor 								:= sWHITE;
	stStatusBanner.sBannerTextColor 							:= sGREEN;
END_IF

(* SYSTEM AUTO CYCLE *)
IF stMachineStatus.bAutoCycle THEN	
	stStatusBanner.sMachineStatusText 							:= 'SYSTEM AUTO CYCLE';		
	stStatusBanner.nMachineStatusColour 						:= nGREEN;
	stStatusBanner.nMachineStatusTxtCol 						:= nWHITE;
	stStatusBanner.sBannerBckColor 								:= sGREEN;
	stStatusBanner.sBannerTextColor 							:= sWHITE;	
END_IF

(* STOPPING *)
IF stMachineStatus.bStopping AND stPuls.bFlash1Hz THEN	
	stStatusBanner.sMachineStatusText 							:= 'STOPPING';		
	stStatusBanner.nMachineStatusColour 						:= nBLACK;
	stStatusBanner.nMachineStatusTxtCol 						:= nWHITE;
	stStatusBanner.sBannerBckColor 								:= sBLACK;
	stStatusBanner.sBannerTextColor 							:= sWHITE;	
ELSIF stMachineStatus.bStopping AND NOT stPuls.bFlash1Hz THEN	
	stStatusBanner.sMachineStatusText 							:= 'STOPPING';		
	stStatusBanner.nMachineStatusColour 						:= nWHITE;
	stStatusBanner.nMachineStatusTxtCol 						:= nBLACK;
	stStatusBanner.sBannerBckColor 								:= sWHITE;
	stStatusBanner.sBannerTextColor 							:= sBLACK;	
END_IF

(*STOPPED *)
IF stMachineStatus.bStopped THEN	
	stStatusBanner.sMachineStatusText 							:= 'CYCLE STOPPED';		
	stStatusBanner.nMachineStatusColour 						:= nBLACK;
	stStatusBanner.nMachineStatusTxtCol 						:= nWHITE;
	stStatusBanner.sBannerBckColor 								:= sBLACK;
	stStatusBanner.sBannerTextColor 							:= sWHITE;	
END_IF

(* FAULT FLASH ON *)
IF stMachineStatus.bFault AND stPuls.bFlash1Hz THEN	
	stStatusBanner.sMachineStatusText 							:= 'FAULT';		
	stStatusBanner.nMachineStatusColour 						:= nRED;
	stStatusBanner.nMachineStatusTxtCol 						:= nWHITE;
	stStatusBanner.sBannerBckColor 								:= sRED;
	stStatusBanner.sBannerTextColor 							:= sWHITE;	
ELSIF stMachineStatus.bFault AND NOT stPuls.bFlash1Hz THEN	
	stStatusBanner.sMachineStatusText 							:= 'FAULT';		
	stStatusBanner.nMachineStatusColour 						:= nWHITE;
	stStatusBanner.nMachineStatusTxtCol 						:= nBLACK;
	stStatusBanner.sBannerBckColor 								:= sWHITE;
	stStatusBanner.sBannerTextColor 							:= sBLACK;	
END_IF

(* MANUAL MODE *)
IF stMachineStatus.bManualMode THEN	
	stStatusBanner.sMachineStatusText 							:= 'MANUAL MODE';		
	stStatusBanner.nMachineStatusColour 						:= nBLUE;
	stStatusBanner.nMachineStatusTxtCol 						:= nWHITE;
	stStatusBanner.sBannerBckColor 								:= sBLUE;
	stStatusBanner.sBannerTextColor 							:= sWHITE;	
END_IF
END_ACTION

ACTION b_ACT_Timers:

stTimers.tAutoCycleTimeOut		:= DINT_TO_TIME(stTimers.nAutoCycleTimeOut * 1000) ;
stTimers.tDoorOpenedSignal		:= DINT_TO_TIME(stTimers.nDoorOpenedSignal * 1000) ;
stTimers.tStation1TimeOut		:= DINT_TO_TIME(stTimers.nStation1TimeOut * 1000) ;
stTimers.tStation2TimeOut		:= DINT_TO_TIME(stTimers.nStation2TimeOut * 1000) ;
stTimers.tStation3TimeOut		:= DINT_TO_TIME(stTimers.nStation3TimeOut * 1000) ;
stTimers.tTwoHandsSignal		:= DINT_TO_TIME(stTimers.nTwoHandsSignal * 1000) ;
stTimers.tHeightTest			:= DINT_TO_TIME(stTimers.nHeightTest * 1000) ;
stTimers.tAutoCycleIDLETimeOut			:= DINT_TO_TIME(stTimers.nAutoCycleIDLETimeOut * 1000) ;
END_ACTION

ACTION c_ACT_IO:
dw_T09_EL2809.qPanelLightLED				:= bLightsOnOff;
END_ACTION

END_PROGRAM

// ---- POUs/B_STATIONS/B_1_LEAK_TEST/B_1_1_PRG_Master_Leak_Test.TcPOU
PROGRAM B_1_1_PRG_Master_Leak_Test

VAR

	tonStationStopped					: TON;
	tonExecute							: TON;
	rGoodStatistics						: ARRAY [0..1] OF R_TRIG;
	rBadStatistics						: ARRAY [0..1] OF R_TRIG;
	rEfficency							: ARRAY [0..1] OF STRING(510);
	
	tonWaitResults						: TON;
/////////////////////////////////////////////////////////////////////////////////////I O/////////////////////////////////////////////////////////////////////////////////////	

	bStopped							: ARRAY [0..1] OF BOOL;
	bError								: ARRAY [0..1] OF BOOL;
	bReady								: ARRAY [0..1] OF BOOL;
	bDone								: ARRAY [0..1] OF BOOL;
	bReset								: ARRAY [0..1] OF BOOL;
	bStart								: ARRAY [0..1] OF BOOL;
	bStop								: ARRAY [0..1] OF BOOL;	
	bBusy								: ARRAY [0..1] OF BOOL;	
	fLeakTestDone						: ARRAY [0..1] OF F_TRIG;	
	bLeakTestDone						: ARRAY [0..1] OF BOOL;	
	rPass								: ARRAY [0..1] OF R_TRIG;	
	bPass								: ARRAY [0..1] OF BOOL;	
	rFail								: ARRAY [0..1] OF R_TRIG;	
	bFail								: ARRAY [0..1] OF BOOL;
	rReset								: ARRAY [0..1] OF R_TRIG;
	
END_VAR

a_ACT_Ctrl_Station_1();
b_ACT_IO();
c_ACT_Statistics_Station_1();
d_ACT_Set_Events_Station_1();

ACTION a_ACT_Ctrl_Station_1:
/////////////////////////////////////////////////////////////////////////////////////UTILITIES/////////////////////////////////////////////////////////////////////////////////////
tonStationStopped( IN := bStopped[0] AND bStopped[1], PT := T#1S);
tonExecute(IN := stLeakTesters.State = E_LeakTester_State.RUN_LEAK_TESTERS, PT := T#500MS);
tonWaitResults(IN := (stLeakTesters.State = E_LeakTester_State.WAIT_RESULTS), PT := T#100MS);

/////////////////////////////////////////////////////////////////////////////////////CONDITIONS/////////////////////////////////////////////////////////////////////////////////////

IF stLeakTesters.CMD.bAbort OR bError[0] OR bError[1] THEN
								
	stLeakTesters.State											:= E_LeakTester_State.RESET;
	

END_IF



CASE stLeakTesters.State OF
	
	E_LeakTester_State.ABORTED:
	
								IF stLeakTesters.CMD.bEnable AND NOT bError[0] THEN
									stLeakTesters.State			:= E_LeakTester_State.HOMING;
								ELSIF bError[0] OR bError[1] THEN
									stLeakTesters.State			:= E_LeakTester_State.ERROR;
								END_IF
	
	E_LeakTester_State.HOMING:
	
								IF bReady[0] AND bReady[1] AND bStopped[0] AND bStopped[1] THEN
									stLeakTesters.State			:= E_LeakTester_State.READY;
								
								END_IF
								
	E_LeakTester_State.READY:
	
								IF stLeakTesters.CMD.bExecute THEN
									
									stLeakTesters.State			:= E_LeakTester_State.RUN_LEAK_TESTERS;
								
								END_IF
		
								
	E_LeakTester_State.RUN_LEAK_TESTERS:	
								
								IF stLeakTesters.CMD.LeakTestersCMD.RunLeakTester1 AND stLeakTesters.CMD.LeakTestersCMD.RunLeakTester2 THEN
										
										bStart[0]				:= TRUE;
										bStart[1]				:= TRUE;
									
								ELSIF stLeakTesters.CMD.LeakTestersCMD.RunLeakTester1 AND NOT stLeakTesters.CMD.LeakTestersCMD.RunLeakTester2 THEN
										
										bStart[0]				:= TRUE;
									
								ELSIF NOT stLeakTesters.CMD.LeakTestersCMD.RunLeakTester1 AND stLeakTesters.CMD.LeakTestersCMD.RunLeakTester2 THEN
										
										bStart[1]				:= TRUE;
									
								END_IF
								
								IF tonExecute.Q THEN
									
									stLeakTesters.State			:= E_LeakTester_State.WAIT_LEAK_TESTERS;
								
								END_IF
	
	E_LeakTester_State.WAIT_LEAK_TESTERS:
	
								IF stLeakTesters.CMD.LeakTestersCMD.RunLeakTester1 AND stLeakTesters.CMD.LeakTestersCMD.RunLeakTester2 THEN
										
										IF bLeakTestDone[0] AND bLeakTestDone[1] THEN
											
											stLeakTesters.State	:= E_LeakTester_State.WAIT_RESULTS;
											
										END_IF
									
								ELSIF stLeakTesters.CMD.LeakTestersCMD.RunLeakTester1 AND NOT stLeakTesters.CMD.LeakTestersCMD.RunLeakTester2 THEN
										
										IF bLeakTestDone[0]  THEN
											
											stLeakTesters.State	:= E_LeakTester_State.WAIT_RESULTS;
											
										END_IF
									
								ELSIF NOT stLeakTesters.CMD.LeakTestersCMD.RunLeakTester1 AND stLeakTesters.CMD.LeakTestersCMD.RunLeakTester2 THEN
										
										IF bLeakTestDone[1]  THEN
											
											stLeakTesters.State	:= E_LeakTester_State.WAIT_RESULTS;
											
										END_IF
									
								END_IF
	
	E_LeakTester_State.WAIT_RESULTS:
	
								IF tonWaitResults.Q THEN
									
									stLeakTesters.State	:= E_LeakTester_State.RESULTS;
									
								END_IF


		
	E_LeakTester_State.RESULTS:
								
								IF stLeakTesters.CMD.LeakTestersCMD.RunLeakTester1 THEN
									
									IF bPass[0] THEN
									
										stCycleDataNest1.LeakTest_Pass := TRUE;
										stCycleDataNest1.LeakTest_Fail := FALSE;
										
										stLeakTesters.State	:= E_LeakTester_State.DONE;
								
									ELSIF bFail[0] THEN
									
										stCycleDataNest1.LeakTest_Fail := TRUE;
										stCycleDataNest1.LeakTest_Pass := FALSE;
								
										stLeakTesters.State	:= E_LeakTester_State.DONE;
										
								END_IF
									
								END_IF
								
								IF stLeakTesters.CMD.LeakTestersCMD.RunLeakTester2 THEN
									
									IF bPass[1] THEN
									
										stCycleDataNest2.LeakTest_Pass := TRUE;
										stCycleDataNest2.LeakTest_Fail	:= FALSE;
										
										stLeakTesters.State	:= E_LeakTester_State.DONE;
								
									ELSIF bFail[1] THEN
									
										stCycleDataNest2.LeakTest_Fail	:= TRUE;
										stCycleDataNest2.LeakTest_Pass := FALSE;
										
										stLeakTesters.State	:= E_LeakTester_State.DONE;
								
								END_IF
									
								END_IF
								
								
								
		E_LeakTester_State.DONE:
								IF  stLeakTesters.CMD.bAcknowledge THEN
									
									stLeakTesters.CMD.bAcknowledge := FALSE;
									stLeakTesters.State			:= E_LeakTester_State.RESET;
									
								END_IF	
								
								
								
	E_LeakTester_State.RESET:
	

								bStart[0]						:= FALSE;
								bStart[1]						:= FALSE;
								bReset[0]						:= FALSE;
								bReset[1]						:= FALSE;
								bStop[0]						:= FALSE;
								bStop[1]						:= FALSE;
								bLeakTestDone[0]				:= FALSE;
								bLeakTestDone[1]				:= FALSE;
								bPass[0]						:= FALSE;
								bPass[1]						:= FALSE;
								bFail[0]						:= FALSE;
								bFail[1]						:= FALSE;
								
								IF bError[0] OR bError[1] THEN

									stLeakTesters.State		:= E_LeakTester_State.ERROR;

								ELSIF stLeakTesters.CMD.bAbort OR stLeakTesters.CMD.bEndCycle THEN
									
									stLeakTesters.State			:= E_LeakTester_State.ABORTED;
									
								ELSE stLeakTesters.State			:= E_LeakTester_State.READY;
								
								END_IF
								
								
								
	E_LeakTester_State.STOPPING: 
	
								bStop[0]						:= TRUE;
								bStop[1]						:= TRUE;
								
								IF tonStationStopped.Q THEN
									
									stLeakTesters.State			:= E_LeakTester_State.RESET;
									
								END_IF
	
	E_LeakTester_State.ERROR:
	
								IF NOT bError[0] AND bError[1] THEN
									
									stLeakTesters.State						:= E_LeakTester_State.ABORTED;
									
								END_IF

ELSE stLeakTesters.State := E_LeakTester_State.ABORTED;
	
END_CASE
/////////////////////////////////////////////////////////////////////////////////////STATUS/////////////////////////////////////////////////////////////////////////////////////

stLeakTesters.Status.bBusy	:= 	stLeakTesters.State = E_LeakTester_State.STOPPING OR
								stLeakTesters.State = E_LeakTester_State.HOMING OR
								stLeakTesters.State = E_LeakTester_State.RUN_LEAK_TESTERS OR
								stLeakTesters.State = E_LeakTester_State.WAIT_LEAK_TESTERS;

stLeakTesters.Status.bDone	:= 	stLeakTesters.State = E_LeakTester_State.DONE;

stLeakTesters.Status.bError	:= 	stLeakTesters.State = E_LeakTester_State.ERROR;	

stLeakTesters.Status.bReady	:=	stLeakTesters.State = E_LeakTester_State.READY;

stLeakTesters.Status.bStopped := NOT stLeakTesters.Status.bBusy;
END_ACTION

ACTION b_ACT_IO:


bStopped[0]								:= NOT LeakTester1_IO.sti28General_I_O.bTestActiveLiveData;
bStopped[1]								:= NOT LeakTester2_IO.sti28General_I_O.bTestActiveLiveData;
bError[0]								:= LeakTester1_IO.sti28General_I_O.bMalfunction;
bError[1]								:= LeakTester2_IO.sti28General_I_O.bMalfunction;
bReady[0]								:= LeakTester1_IO.sti28General_I_O.bInstrumentReady;
bReady[1]								:= LeakTester2_IO.sti28General_I_O.bInstrumentReady;
LeakTester1_IO.sti28General_I_O.bReset	:= bReset[0] OR bLeaktester1_Reset;	
LeakTester2_IO.sti28General_I_O.bReset	:= bReset[1] OR bLeaktester2_Reset;	
LeakTester1_IO.sti28General_I_O.bStart	:= bStart[0] OR bLeaktester1_Start;
LeakTester2_IO.sti28General_I_O.bStart	:= bStart[1] OR bLeaktester2_Start;
LeakTester1_IO.sti28General_I_O.bStop	:= bStop[0] OR bLeaktester1_Stop OR stLeakTesters.CMD.bAbort;
LeakTester2_IO.sti28General_I_O.bStop	:= bStop[1] OR bLeaktester2_Stop OR stLeakTesters.CMD.bAbort;



rReset[0](CLK := stLeakTesters.CMD.bReset, Q => bReset[0]);
rReset[1](CLK := stLeakTesters.CMD.bReset, Q => bReset[1]);

fLeakTestDone[0](CLK := LeakTester1_IO.sti28General_I_O.bTestActiveLiveData);
fLeakTestDone[1](CLK := LeakTester2_IO.sti28General_I_O.bTestActiveLiveData);
rPass[0](CLK := LeakTester1_IO.sti28General_I_O.bProgramAccept);
rPass[1](CLK := LeakTester2_IO.sti28General_I_O.bProgramAccept);
rFail[0](CLK := LeakTester1_IO.sti28General_I_O.bProgramReject);
rFail[1](CLK := LeakTester2_IO.sti28General_I_O.bProgramReject);



IF fLeakTestDone[0].Q THEN
	
	bLeakTestDone[0]					:= TRUE;
	
END_IF

IF fLeakTestDone[1].Q THEN
	
	bLeakTestDone[1]					:= TRUE;
	
END_IF

IF rPass[0].Q THEN
	
	bPass[0]							:= TRUE;

END_IF

IF rPass[1].Q THEN
	
	bPass[1]							:= TRUE;

END_IF

IF rFail[0].Q THEN
	
	bFail[0]							:= TRUE;

END_IF

IF rFail[1].Q THEN
	
	bFail[1]							:= TRUE;

END_IF
END_ACTION

ACTION c_ACT_Statistics_Station_1:
stStatisticsHMI[2].sName			:= 'LEAK TESTER 1';
stStatisticsHMI[3].sName			:= 'LEAK TESTER 2';


rGoodStatistics[0]( CLK := stCycleDataNest1.LeakTest_Pass );
rGoodStatistics[1]( CLK := stCycleDataNest2.LeakTest_Pass );
rBadStatistics[0] ( CLK := stCycleDataNest1.LeakTest_Fail );
rBadStatistics[1] ( CLK := stCycleDataNest2.LeakTest_Fail );

IF 	rGoodStatistics[0].Q THEN
	
	stStatisticsHMI[2].nGood		:= stStatisticsHMI[2].nGood + 1;
	
END_IF
								
IF 	rBadStatistics[0].Q THEN
	
	stStatisticsHMI[2].nBad			:= stStatisticsHMI[2].nBad + 1;
	
END_IF

IF stStatisticsHMI[2].bResetGood THEN
	stStatisticsHMI[2].nGood		:= 0;
END_IF

IF stStatisticsHMI[2].bResetBad THEN
	stStatisticsHMI[2].nBad			:= 0;
END_IF


IF 	rGoodStatistics[1].Q THEN
	
	stStatisticsHMI[3].nGood		:= stStatisticsHMI[3].nGood + 1;
	
END_IF
								
IF 	rBadStatistics[1].Q THEN
	
	stStatisticsHMI[3].nBad			:= stStatisticsHMI[3].nBad + 1;
	
END_IF

IF stStatisticsHMI[3].bResetGood THEN
	stStatisticsHMI[3].nGood		:= 0;
END_IF

IF stStatisticsHMI[3].bResetBad THEN
	stStatisticsHMI[3].nBad			:= 0;
END_IF



IF (( stStatisticsHMI[2].nGood + stStatisticsHMI[2].nBad) <> 0) THEN
	
	rEfficency[0]							:= LREAL_TO_FMTSTR(in := (DINT_TO_REAL(stStatisticsHMI[2].nGood) /( DINT_TO_REAL(stStatisticsHMI[2].nGood) + DINT_TO_REAL(stStatisticsHMI[2].nBad))) * 100.0,iPrecision := 2, bRound := TRUE);
	stStatisticsHMI[2].nEfficency		:= CONCAT(STR1 := '%', STR2 := (rEfficency[0]));

ELSE stStatisticsHMI[2].nEfficency		:= CONCAT(STR1 := '%', STR2 := (DINT_TO_STRING(0)));
	
END_IF

IF (( stStatisticsHMI[3].nGood + stStatisticsHMI[3].nBad) <> 0) THEN
	
	rEfficency[1]							:= LREAL_TO_FMTSTR(in := (DINT_TO_REAL(stStatisticsHMI[3].nGood) /( DINT_TO_REAL(stStatisticsHMI[3].nGood) + DINT_TO_REAL(stStatisticsHMI[3].nBad))) * 100.0,iPrecision := 2, bRound := TRUE);
	stStatisticsHMI[3].nEfficency		:= CONCAT(STR1 := '%', STR2 := (rEfficency[1]));

ELSE stStatisticsHMI[3].nEfficency		:= CONCAT(STR1 := '%', STR2 := (DINT_TO_STRING(0)));
	
END_IF
END_ACTION

ACTION d_ACT_Set_Events_Station_1:
//IMMEDIATE FAULTS

stStationEvents[1].aEvents[0].bFault						:= TRUE;
stStationEvents[1].aEvents[0].bEventTimer( IN := (stLeakTesters.State = E_LeakTester_State.RUN_LEAK_TESTERS) OR (stLeakTesters.State = E_LeakTester_State.WAIT_LEAK_TESTERS), PT := stTimers.tStation1TimeOut);
stStationEvents[1].aEvents[0].bEventFlag					:= stStationEvents[1].aEvents[0].bEventTimer.Q;
stStationEvents[1].aEvents[0].bEventText					:= 'Leak tester cycle Timeout';
stStationEvents[1].aEvents[0].sSolution						:= 'Reset System';



//CYCLE STOP REQUEST

stStationEvents[1].aEvents[20].bCycleStopRequest				:= TRUE;
stStationEvents[1].aEvents[20].bEventFlag					:= NOT bReady[0] AND (stLeakTesters.State = E_LeakTester_State.HOMING);// AND (stLeakTesters.State = E_LeakTester_State.HOMING);
stStationEvents[1].aEvents[20].bEventText					:= 'Leak Tester 1 not ready';
stStationEvents[1].aEvents[20].sSolution						:= 'Check Leak tester 1';

stStationEvents[1].aEvents[21].bCycleStopRequest				:= TRUE;
stStationEvents[1].aEvents[21].bEventFlag					:= NOT bReady[1] AND (stLeakTesters.State = E_LeakTester_State.HOMING);// AND (stLeakTesters.State = E_LeakTester_State.HOMING);
stStationEvents[1].aEvents[21].bEventText					:= 'Leak Tester 2 not ready';
stStationEvents[1].aEvents[21].sSolution						:= 'Check Leak tester 2';

stStationEvents[1].aEvents[22].bCycleStopRequest			:= TRUE;
stStationEvents[1].aEvents[22].bEventFlag					:= bError[0] AND bNest1Flag;
stStationEvents[1].aEvents[22].bEventText					:= 'Leak Tester 1 malfunction';
stStationEvents[1].aEvents[22].sSolution					:= 'Check Leak tester 1';

stStationEvents[1].aEvents[23].bCycleStopRequest			:= TRUE;
stStationEvents[1].aEvents[23].bEventFlag					:=  bError[1] AND bNest2Flag;
stStationEvents[1].aEvents[23].bEventText					:= 'Leak Tester 2 malfunction';
stStationEvents[1].aEvents[23].sSolution					:= 'Check Leak tester 2';

stStationEvents[1].aEvents[24].bCycleStopRequest			:= TRUE;
stStationEvents[1].aEvents[24].rEventTrigger( CLK := LeakTester1_IO.sti28LasResult.inPartEvaluation = 13);
stStationEvents[1].aEvents[24].bEventFlag					:=  stStationEvents[1].aEvents[24].rEventTrigger.Q;
stStationEvents[1].aEvents[24].bEventText					:= 'Leak Tester 1 Low Pressure';
stStationEvents[1].aEvents[24].sSolution					:= 'Check Leak tester 1 pneumatic circuit ';

stStationEvents[1].aEvents[25].bCycleStopRequest			:= TRUE;
stStationEvents[1].aEvents[25].rEventTrigger( CLK := LeakTester1_IO.sti28LasResult.inPartEvaluation = 14);
stStationEvents[1].aEvents[25].bEventFlag					:=  stStationEvents[1].aEvents[25].rEventTrigger.Q;
stStationEvents[1].aEvents[25].bEventText					:= 'Leak Tester 1 High Pressure';
stStationEvents[1].aEvents[25].sSolution					:= 'Check Leak tester 1 parameters';

stStationEvents[1].aEvents[26].bCycleStopRequest			:= TRUE;
stStationEvents[1].aEvents[26].rEventTrigger( CLK := LeakTester2_IO.sti28LasResult.inPartEvaluation = 13);
stStationEvents[1].aEvents[26].bEventFlag					:=  stStationEvents[1].aEvents[26].rEventTrigger.Q;
stStationEvents[1].aEvents[26].bEventText					:= 'Leak Tester 2 Low Pressure';
stStationEvents[1].aEvents[26].sSolution					:= 'Check Leak tester 2 pneumatic circuit ';

stStationEvents[1].aEvents[27].bCycleStopRequest			:= TRUE;
stStationEvents[1].aEvents[27].rEventTrigger( CLK := LeakTester2_IO.sti28LasResult.inPartEvaluation = 14);
stStationEvents[1].aEvents[27].bEventFlag					:=  stStationEvents[1].aEvents[27].rEventTrigger.Q;
stStationEvents[1].aEvents[27].bEventText					:= 'Leak Tester 2 High Pressure';
stStationEvents[1].aEvents[27].sSolution					:= 'Check Leak tester 2 parameters';


//Message
(*
stStationEvents[1].aEvents[3].bMessage						:= TRUE;
stStationEvents[1].aEvents[3].bEventFlag					:= bEventsFlag[3];
stStationEvents[1].aEvents[3].bEventText					:= 'Message 3';
stStationEvents[1].aEvents[3].sSolution						:= '';*)
END_ACTION

END_PROGRAM

// ---- POUs/B_STATIONS/B_4_PROCESS_CYLINDER__SLIDE_DOOR_SLIDE_NEST/B_4_1_PRG_Master_ProcessCylinder.TcPOU
PROGRAM B_4_1_PRG_Master_ProcessCylinder

VAR

	
	
/////////////////////////////////////////////////////////////////////////////////////I O/////////////////////////////////////////////////////////////////////////////////////	
	bExtended							: BOOL;
	bRetracted							: BOOL;
	bExtend								: BOOL;
	bRetract							: BOOL;
	
	bProcessDoorClosed					: BOOL;
	
END_VAR

d_ACT_Set_Events_Station_4A();
a_ACT_Ctrl_Station_4A();
b_ACT_IO_A();
c_Manual();

ACTION a_ACT_Ctrl_Station_4A:
/////////////////////////////////////////////////////////////////////////////////////UTILITIES/////////////////////////////////////////////////////////////////////////////////////

/////////////////////////////////////////////////////////////////////////////////////CONDITIONS/////////////////////////////////////////////////////////////////////////////////////


IF stProcessCylinder.CMD.bAbort THEN
	
	stProcessCylinder.State				:= E_ProcessCylinder_State.RESET;

END_IF

CASE stProcessCylinder.State OF
	
	E_ProcessCylinder_State.ABORTED:
	
								IF stProcessCylinder.CMD.bEnable THEN
									
									stProcessCylinder.State				:= E_ProcessCylinder_State.HOMING;
								
								END_IF
								
	E_ProcessCylinder_State.HOMING:
	
								IF bProcessDoorClosed THEN
									
									bRetract							:= TRUE;
									
								END_IF
								
								
								IF bRetracted THEN
									
									bRetract							:= FALSE;
									stProcessCylinder.State				:= E_ProcessCylinder_State.READY;
									
								
								END_IF
	
	E_ProcessCylinder_State.READY:
	
								IF stProcessCylinder.CMD.bExecute AND stProcessCylinder.CMD.ProcessCylinderCMD.ExtendCylinder THEN

									stProcessCylinder.State				:= E_ProcessCylinder_State.EXTEND;
									
								ELSIF stProcessCylinder.CMD.bExecute AND stProcessCylinder.CMD.ProcessCylinderCMD.RetractCylinder THEN
									
									stProcessCylinder.State				:= E_ProcessCylinder_State.RETRACT;;									
																		
								END_IF
	
	E_ProcessCylinder_State.EXTEND:
	
								bExtend									:= stProcessCylinder.CMD.ProcessCylinderCMD.ExtendCylinder;
								
								IF bExtend THEN
									
									IF bExtended THEN

										stProcessCylinder.State			:= E_ProcessCylinder_State.DONE;
									
									END_IF						
	
								END_IF
								
	E_ProcessCylinder_State.RETRACT:
	
								bRetract								:= stProcessCylinder.CMD.ProcessCylinderCMD.RetractCylinder;
								
								
								IF bRetract THEN
									
									IF bRetracted THEN

										stProcessCylinder.State				:= E_ProcessCylinder_State.DONE;
									
									END_IF					
	
								END_IF
								
	E_ProcessCylinder_State.DONE:
	
								IF stProcessCylinder.CMD.bAcknowledge THEN
									
									stProcessCylinder.CMD.bAcknowledge		:= FALSE;
									stProcessCylinder.State					:= E_ProcessCylinder_State.RESET;
								
								END_IF
	
	
	E_ProcessCylinder_State.RESET:	
	
								bExtend										:= FALSE;								
								bRetract									:= FALSE;
								
								
								IF NOT stProcessCylinder.CMD.bAbort AND NOT stProcessCylinder.CMD.bEndCycle THEN
									
									stProcessCylinder.State					:= E_ProcessCylinder_State.READY;
									
								ELSE stProcessCylinder.State					:= E_ProcessCylinder_State.ABORTED;
								END_IF
									

ELSE stProcessCylinder.State	:= E_ProcessCylinder_State.ABORTED;
	
END_CASE
/////////////////////////////////////////////////////////////////////////////////////STATUS/////////////////////////////////////////////////////////////////////////////////////

stProcessCylinder.Status.bBusy		:= 	stProcessCylinder.State	= E_ProcessCylinder_State.EXTEND OR
										stProcessCylinder.State	= E_ProcessCylinder_State.RETRACT OR 
										stProcessCylinder.State	= E_ProcessCylinder_State.STOPPING;
								
stProcessCylinder.Status.bDone		:=	stProcessCylinder.State	= E_ProcessCylinder_State.DONE;

stProcessCylinder.Status.bReady		:= 	stProcessCylinder.State	= E_ProcessCylinder_State.READY;

stProcessCylinder.Status.bStopped	:= 	NOT stProcessCylinder.Status.bBusy;
END_ACTION

ACTION b_ACT_IO_A:

bExtended								:= dw_T08_EL1809.iProcessCylinderExtended;
bRetracted								:= stTwinSAFE.qProcessCylinderRetracted;

IF bExtend OR bProcessCylinderDown AND (dw_T08_EL1809.iSlideNestExtended OR dw_T08_EL1809.iSlideNestRetracted) THEN
	
	dw_T09_EL2809.qExtendProcessCylinder	:= TRUE ;
	dw_T09_EL2809.qRetractProcessCylinder	:= FALSE;

ELSIF bRetract OR bProcessCylinder_Up THEN
	
	dw_T09_EL2809.qExtendProcessCylinder	:= FALSE;
	dw_T09_EL2809.qRetractProcessCylinder	:= TRUE;
	
ELSIF stMachineStatus.bFault THEN
	
	dw_T09_EL2809.qExtendProcessCylinder	:= FALSE;
	dw_T09_EL2809.qRetractProcessCylinder	:= FALSE;

END_IF


IF stStationEvents[3].aEvents[0].bEventTimer.Q THEN
	
	bRetract := FALSE;

END_IF

IF stStationEvents[3].aEvents[1].bEventTimer.Q THEN
	
	bExtended := FALSE;

END_IF

bProcessDoorClosed := dw_T05_EL1918.iProcessDoorClosed1 AND dw_T05_EL1918.iProcessDoorClosed2 AND dw_T05_EL1918.iProcessDoorFB;
END_ACTION

ACTION c_Manual:
(*
IF bProcessCylinder1_Up THEN
	
	bRetract[0] := TRUE;
	
ELSIF bRetracted[0] THEN
	
	bRetract[0] := FALSE;

END_IF

IF bProcessCylinder1_Down THEN
	
	bExtend[0] := TRUE;
	
ELSIF bExtended[0] THEN
	
	bExtend[0] := FALSE;

END_IF

IF bProcessCylinder2_Up THEN
	
	bRetract[1] := TRUE;
	
ELSIF bRetracted[1] THEN
	
	bRetract[1] := FALSE;

END_IF

IF bProcessCylinder2_Down THEN
	
	bExtend[1] := TRUE;
	
ELSIF bExtended[1] THEN
	
	bExtend[1] := FALSE;

END_IF
*)
END_ACTION

ACTION d_ACT_Set_Events_Station_4A:
//FAULTS

stStationEvents[3].aEvents[0].bEventTimer( IN := (bExtend AND NOT bExtended), PT := T#10S);
stStationEvents[3].aEvents[0].bFault						:= TRUE;
stStationEvents[3].aEvents[0].bEventFlag					:= stStationEvents[3].aEvents[0].bEventTimer.Q;
stStationEvents[3].aEvents[0].bEventText					:= 'Process Cylinder 1 extend timeout';
stStationEvents[3].aEvents[0].sSolution						:= 'Check cylinder, neumatic connections and sensors';

stStationEvents[3].aEvents[1].bEventTimer( IN := (bRetract AND NOT bRetracted), PT := T#3S);
stStationEvents[3].aEvents[1].bFault						:= TRUE;
stStationEvents[3].aEvents[1].bEventFlag					:= stStationEvents[3].aEvents[1].bEventTimer.Q;
stStationEvents[3].aEvents[1].bEventText					:= 'Process Cylinder retract timeout';
stStationEvents[3].aEvents[1].sSolution						:= 'Check cylinder, neumatic connections and sensors';


//CYCLE STOP REQUEST

(*stStationEvents[3].aEvents[2].bCycleStopRequest			:= TRUE;
stStationEvents[3].aEvents[2].bEventFlag					:= ;
stStationEvents[3].aEvents[2].bEventText					:= 'ST1 EVENT 7';*)
END_ACTION

END_PROGRAM

// ---- POUs/B_STATIONS/B_4_PROCESS_CYLINDER__SLIDE_DOOR_SLIDE_NEST/B_4_2_PRG_Master_ProcessDoor.TcPOU
PROGRAM B_4_2_PRG_Master_ProcessDoor

VAR

	bEventsFlag							: ARRAY [0..100] OF BOOL;
/////////////////////////////////////////////////////////////////////////////////////I O/////////////////////////////////////////////////////////////////////////////////////	
	
	bOpenDoor							: BOOL;
	bCloseDoor							: BOOL;
	bCloseDoorHMI						: BOOL;
	bOpenDoorHMI						: BOOL;
	bDoorClosed							: BOOL;
	tonDoorOpened						: TON;
	bDoorOpened							: BOOL;
	
	bProcessCylinderNotHomed			: BOOL;
	bSlideNestNotHomed					: BOOL;
	
	

	
	
END_VAR

d_ACT_Set_Events_Station_4B();
a_ACT_Ctrl_Station_4B();
b_ACT_IO_B();
c_Manual();

ACTION a_ACT_Ctrl_Station_4B:
/////////////////////////////////////////////////////////////////////////////////////UTILITIES/////////////////////////////////////////////////////////////////////////////////////

/////////////////////////////////////////////////////////////////////////////////////CONDITIONS/////////////////////////////////////////////////////////////////////////////////////
IF stProcessDoor.State <> E_ProcessDoor_State.HOMING THEN
	
	bDoorClosingInitFlag											:= FALSE;

END_IF


IF stProcessDoor.CMD.bAbort THEN
	
	stProcessDoor.State				:= E_ProcessDoor_State.RESET;
	
ELSIF stProcessDoor.CMD.bEndCycle THEN
	
	stProcessDoor.State				:= E_ProcessDoor_State.STOPPING;

END_IF

CASE stProcessDoor.State OF
	
	E_ProcessDoor_State.ABORTED:
	
								IF stProcessDoor.CMD.bEnable THEN
									
									stProcessDoor.State				:= E_ProcessDoor_State.HOMING;
								
								END_IF
								
		E_ProcessDoor_State.HOMING: 
		
								IF bProcessCylinderNotHomed OR bSlideNestNotHomed THEN
									
									bCloseDoor						:= TRUE;
									bOpenDoor						:= FALSE;
									
									IF NOT bDoorClosed AND bCloseDoor THEN
										
										bDoorClosingInitFlag		:= TRUE;
									ELSE bDoorClosingInitFlag		:= FALSE;
									END_IF
									
								ELSE
									
									bCloseDoor						:= FALSE;
									bOpenDoor						:= TRUE;
									
								END_IF
								
								IF bDoorOpened AND NOT (bProcessCylinderNotHomed OR bSlideNestNotHomed) THEN
									
									stProcessDoor.State				:= E_ProcessDoor_State.READY;									
									bOpenDoor						:= FALSE;
																	
								END_IF
	
	
	E_ProcessDoor_State.READY:
	
								IF stProcessDoor.CMD.bExecute AND 	stProcessDoor.CMD.ProcessDoorCMD.OpenDoor	THEN

									stProcessDoor.State				:= E_ProcessDoor_State.OPEN;
									
								ELSIF stProcessDoor.CMD.bExecute AND 	stProcessDoor.CMD.ProcessDoorCMD.CloseDoor	THEN
									
									stProcessDoor.State				:= E_ProcessDoor_State.CLOSE;									
																		
								END_IF
	

	E_ProcessDoor_State.OPEN:
	
								bOpenDoor							:= TRUE;
								
								IF bDoorOpened	THEN
									
									stProcessDoor.State				:= E_ProcessDoor_State.DONE;
								
								END_IF
								
	E_ProcessDoor_State.CLOSE:
	
								bCloseDoor							:= TRUE;
								
								IF bDoorClosed THEN
									
									stProcessDoor.State				:= E_ProcessDoor_State.DONE;
								
								END_IF
								
	E_ProcessDoor_State.DONE:
	
	
								IF stProcessDoor.CMD.bAcknowledge THEN
									
									stProcessDoor.CMD.bAcknowledge	:= FALSE;
									stProcessDoor.State				:= E_ProcessDoor_State.RESET;
								
								END_IF
	
	
	E_ProcessDoor_State.RESET:	
	
								bOpenDoor							:= FALSE;
								bCloseDoor							:= FALSE;
								
								IF NOT stProcessDoor.CMD.bAbort AND NOT stProcessDoor.CMD.bEndCycle THEN
									
									stProcessDoor.State				:= E_ProcessDoor_State.READY;
									
								ELSE stProcessDoor.State			:= E_ProcessDoor_State.ABORTED;
								END_IF
	
					
	E_ProcessDoor_State.STOPPING:					
									
								bOpenDoor							:= TRUE;
									
								IF bDoorOpened THEN
									
									bOpenDoor						:= FALSE;
									stProcessDoor.State				:= E_ProcessDoor_State.RESET;
								
								END_IF
								
							
														
									

ELSE stProcessDoor.State		:= E_ProcessDoor_State.ABORTED;
	
END_CASE
/////////////////////////////////////////////////////////////////////////////////////STATUS/////////////////////////////////////////////////////////////////////////////////////

stProcessDoor.Status.bBusy			:= 	stProcessDoor.State	= E_ProcessDoor_State.CLOSE OR
										stProcessDoor.State	= E_ProcessDoor_State.OPEN OR 
										stProcessDoor.State	= E_ProcessDoor_State.STOPPING;
								
stProcessDoor.Status.bDone			:=	stProcessDoor.State	= E_ProcessDoor_State.DONE;

stProcessDoor.Status.bReady			:= 	stProcessDoor.State	= E_ProcessDoor_State.READY;

stProcessDoor.Status.bStopped		:= 	NOT stProcessDoor.Status.bBusy;
END_ACTION

ACTION b_ACT_IO_B:
tonDoorOpened( IN := NOT bDoorClosed, PT := stTimers.tDoorOpenedSignal);


bDoorClosed								:= dw_T05_EL1918.iProcessDoorClosed1 AND dw_T05_EL1918.iProcessDoorClosed2 AND dw_T05_EL1918.iProcessDoorFB;
bDoorOpened								:= tonDoorOpened.Q; 
bProcessDoorClosed						:= bDoorClosed;

bDoorOpenedFlag							:= bDoorOpened;

dw_T09_EL2809.qOpenProcessDoor			:= bOpenDoor OR bOpenDoorHMI OR stStationEvents[4].aEvents[0].bEventTimer.Q;//OR bOpenDoorCycleFault;	
dw_T09_EL2809.qCloseProcessDoor			:= bCloseDoor OR bCloseDoorHMI;

bProcessCylinderNotHomed				:= NOT stTwinSAFE.qProcessCylinderRetracted;
bSlideNestNotHomed						:= NOT dw_T08_EL1809.iSlideNestRetracted;
END_ACTION

ACTION c_Manual:


IF bProcessDoor_Down AND stTwinSAFE.qTwoHandsSafe THEN
	
	bCloseDoorHMI					:= TRUE;
	bProcessDoor_Down				:= FALSE;
	
ELSIF bDoorClosed  OR (NOT stMachineStatus.bManualMode AND NOT stMachineStatus.bStopped) THEN

	 bCloseDoorHMI					:= FALSE;
	 bProcessDoor_Down				:= FALSE;

END_IF

IF bProcessDoor_UP THEN
	
	bOpenDoorHMI					:= TRUE;
	
	
ELSIF bDoorOpened OR  (NOT stMachineStatus.bManualMode AND NOT stMachineStatus.bStopped) THEN

	bOpenDoorHMI					:= FALSE;	 
	
END_IF
END_ACTION

ACTION d_ACT_Set_Events_Station_4B:
//IMMEDIATE FAULTS

stStationEvents[4].aEvents[0].bEventTimer( IN :=  (bCloseDoor OR bCloseDoorHMI) AND NOT bDoorClosed, PT := T#2S);
stStationEvents[4].aEvents[0].bFault						:= TRUE;
stStationEvents[4].aEvents[0].bEventFlag					:= stStationEvents[4].aEvents[0].bEventTimer.Q;
stStationEvents[4].aEvents[0].bEventText					:= 'Process Door extend timeout';
stStationEvents[4].aEvents[0].sSolution						:= 'Check cylinder, neumatic connections and sensors';

stStationEvents[4].aEvents[1].bEventTimer( IN :=  (bOpenDoor OR bOpenDoorHMI) AND NOT bDoorOpened, PT := T#2S);
stStationEvents[4].aEvents[1].bFault						:= TRUE;
stStationEvents[4].aEvents[1].bEventFlag					:= stStationEvents[4].aEvents[1].bEventTimer.Q;
stStationEvents[4].aEvents[1].bEventText					:= 'Process Door Retract timeout';
stStationEvents[4].aEvents[1].sSolution						:= 'Check cylinder, neumatic connections and sensors';





//CYCLE STOP REQUEST

(*stStationEvents[4].aEvents[2].bCycleStopRequest			:= TRUE;
stStationEvents[4].aEvents[2].bEventFlag					:= bEventsFlag[2];
stStationEvents[4].aEvents[2].bEventText					:= 'ST1 EVENT 7';*)
END_ACTION

END_PROGRAM

// ---- POUs/B_STATIONS/B_4_PROCESS_CYLINDER__SLIDE_DOOR_SLIDE_NEST/B_4_3_PRG_Master_SlideNest.TcPOU
PROGRAM B_4_3_PRG_Master_SlideNest

VAR


/////////////////////////////////////////////////////////////////////////////////////I O/////////////////////////////////////////////////////////////////////////////////////	
	
	bNestRight							: BOOL;
	bNestLeft							: BOOL;
	bNestRightHMI						: BOOL;
	bLeftRightHMI						: BOOL;
	bNestInLeftPos						: BOOL;
	bNestInRightPos						: BOOL;
	
	bProcessCylinderUp					: BOOL;

	

	
	
END_VAR

d_ACT_Set_Events_Station_4B();
a_ACT_Ctrl_Station_4B();
b_ACT_IO_B();

ACTION a_ACT_Ctrl_Station_4B:
/////////////////////////////////////////////////////////////////////////////////////UTILITIES/////////////////////////////////////////////////////////////////////////////////////

/////////////////////////////////////////////////////////////////////////////////////CONDITIONS/////////////////////////////////////////////////////////////////////////////////////


IF stSlideNest.CMD.bAbort THEN
	
	stSlideNest.State												:= E_SlideNest_State.RESET;
	
ELSIF stSlideNest.CMD.bEndCycle THEN
	
	stSlideNest.State												:= E_SlideNest_State.STOPPING;

END_IF

CASE stSlideNest.State OF
	
	E_SlideNest_State.ABORTED:
	
								IF stSlideNest.CMD.bEnable AND bProcessCylinderUp THEN
									
									stSlideNest.State				:= E_SlideNest_State.HOMING;
								
								END_IF
								
	E_SlideNest_State.HOMING: 
	
								bNestLeft							:= TRUE;
								
								IF bNestInLeftPos THEN
									
